LIN {X 0,Y 368.94,Z 360.526,A -85,B 0,C 180,E1 -12835.146,E2 -12835.146} C_VEL
LIN {X 0,Y 368.933,Z 360.527,A -85,B 0,C 180,E1 -12839.046,E2 -12839.046} C_VEL
LIN {X 0,Y 368.972,Z 360.523,A -85,B 0,C 180,E1 -12842.796,E2 -12842.796} C_VEL
LIN {X 0,Y 368.97,Z 360.526,A -85,B 0,C 180,E1 -12846.421,E2 -12846.421} C_VEL
LIN {X 0,Y 368.94,Z 360.529,A -85,B 0,C 180,E1 -12849.946,E2 -12849.946} C_VEL
LIN {X 0,Y 368.979,Z 360.522,A -85,B 0,C 180,E1 -12853.398,E2 -12853.398} C_VEL
LIN {X 0,Y 369.061,Z 360.512,A -85,B 0,C 180,E1 -12856.789,E2 -12856.789} C_VEL
LIN {X 0,Y 369.07,Z 360.514,A -85,B 0,C 180,E1 -12860.131,E2 -12860.131} C_VEL
LIN {X 0,Y 369.201,Z 360.495,A -85,B 0,C 180,E1 -12863.44,E2 -12863.44} C_VEL
LIN {X 0,Y 369.321,Z 360.481,A -85,B 0,C 180,E1 -12867.818,E2 -12867.818} C_VEL
LIN {X 0,Y 369.46,Z 360.465,A -85,B 0,C 180,E1 -12869.999,E2 -12869.999} C_VEL
LIN {X 0,Y 369.32,Z 360.483,A -85,B 0,C 180,E1 -12872.18,E2 -12872.18} C_VEL
LIN {X 0,Y 369.21,Z 360.493,A -85,B 0,C 180,E1 -12876.557,E2 -12876.557} C_VEL
LIN {X 0,Y 369.138,Z 360.501,A -85,B 0,C 180,E1 -12878.76,E2 -12878.76} C_VEL
LIN {X 0,Y 369.006,Z 360.522,A -85,B 0,C 180,E1 -12882.092,E2 -12882.092} C_VEL
LIN {X 0,Y 369,Z 360.52,A -85,B 0,C 180,E1 -12885.463,E2 -12885.463} C_VEL
LIN {X 0,Y 368.981,Z 360.521,A -85,B 0,C 180,E1 -12888.891,E2 -12888.891} C_VEL
LIN {X 0,Y 368.93,Z 360.528,A -85,B 0,C 180,E1 -12892.394,E2 -12892.394} C_VEL
LIN {X 0,Y 368.997,Z 360.524,A -85,B 0,C 180,E1 -12895.979,E2 -12895.979} C_VEL
LIN {X 0,Y 368.964,Z 360.523,A -85,B 0,C 180,E1 -12898.812,E2 -12898.812} C_VEL
LIN {X 0,Y 368.92,Z 360.531,A -85,B 0,C 180,E1 -12899.621,E2 -12899.621} C_VEL
LIN {X 0,Y 368.255,Z 360.62,A -85,B 0,C 180,E1 -12900.532,E2 -12900.532} C_VEL
LIN {X 0,Y 365.401,Z 360.978,A -85,B 0,C 180,E1 -12902.013,E2 -12902.013} C_VEL
LIN {X 0,Y 362.978,Z 361.275,A -85,B 0,C 180,E1 -12903.21,E2 -12903.21} C_VEL
LIN {X 0,Y 361.934,Z 361.401,A -85,B 0,C 180,E1 -12904.137,E2 -12904.137} C_VEL
LIN {X 0,Y 361.846,Z 361.41,A -85,B 0,C 180,E1 -12904.451,E2 -12904.451} C_VEL
LIN {X 0,Y 361.867,Z 361.408,A -85,B 0,C 180,E1 -12907.224,E2 -12907.224} C_VEL
LIN {X 0,Y 361.899,Z 361.402,A -85,B 0,C 180,E1 -12910.767,E2 -12910.767} C_VEL
LIN {X 0,Y 361.927,Z 361.4,A -85,B 0,C 180,E1 -12914.349,E2 -12914.349} C_VEL
LIN {X 0,Y 361.885,Z 361.408,A -85,B 0,C 180,E1 -12917.557,E2 -12917.557} C_VEL
LIN {X 0,Y 361.868,Z 361.407,A -85,B 0,C 180,E1 -12920.971,E2 -12920.971} C_VEL
LIN {X 0,Y 361.867,Z 361.406,A -85,B 0,C 180,E1 -12924.654,E2 -12924.654} C_VEL
LIN {X 0,Y 361.829,Z 361.411,A -85,B 0,C 180,E1 -12928.37,E2 -12928.37} C_VEL
LIN {X 0,Y 361.893,Z 361.403,A -85,B 0,C 180,E1 -12930.955,E2 -12930.955} C_VEL
LIN {X 0,Y 361.946,Z 361.4,A -85,B 0,C 180,E1 -12933.474,E2 -12933.474} C_VEL
LIN {X 0,Y 361.881,Z 361.406,A -85,B 0,C 180,E1 -12937.144,E2 -12937.144} C_VEL
LIN {X 0,Y 361.912,Z 361.4,A -85,B 0,C 180,E1 -12940.724,E2 -12940.724} C_VEL
LIN {X 0,Y 361.939,Z 361.398,A -85,B 0,C 180,E1 -12944.226,E2 -12944.226} C_VEL
LIN {X 0,Y 361.99,Z 361.391,A -85,B 0,C 180,E1 -12946.528,E2 -12946.528} C_VEL
LIN {X 0,Y 362.026,Z 361.389,A -85,B 0,C 180,E1 -12949.938,E2 -12949.938} C_VEL
LIN {X 0,Y 362.141,Z 361.372,A -85,B 0,C 180,E1 -12952.192,E2 -12952.192} C_VEL
LIN {X 0,Y 362.109,Z 361.376,A -85,B 0,C 180,E1 -12954.431,E2 -12954.431} C_VEL
LIN {X 0,Y 362.274,Z 361.359,A -85,B 0,C 180,E1 -12957.777,E2 -12957.777} C_VEL
LIN {X 0,Y 362.42,Z 361.338,A -85,B 0,C 180,E1 -12960,E2 -12960} C_VEL
LIN {X 0,Y 362.274,Z 361.355,A -85,B 0,C 180,E1 -12962.224,E2 -12962.224} C_VEL
LIN {X 0,Y 362.168,Z 361.368,A -85,B 0,C 180,E1 -12966.686,E2 -12966.686} C_VEL
LIN {X 0,Y 362.066,Z 361.382,A -85,B 0,C 180,E1 -12968.934,E2 -12968.934} C_VEL
LIN {X 0,Y 361.958,Z 361.394,A -85,B 0,C 180,E1 -12972.333,E2 -12972.333} C_VEL
LIN {X 0,Y 361.953,Z 361.395,A -85,B 0,C 180,E1 -12974.621,E2 -12974.621} C_VEL
LIN {X 0,Y 361.946,Z 361.397,A -85,B 0,C 180,E1 -12978.1,E2 -12978.1} C_VEL
LIN {X 0,Y 361.884,Z 361.407,A -85,B 0,C 180,E1 -12981.654,E2 -12981.654} C_VEL
LIN {X 0,Y 361.92,Z 361.405,A -85,B 0,C 180,E1 -12985.291,E2 -12985.291} C_VEL
LIN {X 0,Y 361.9,Z 361.404,A -85,B 0,C 180,E1 -12987.78,E2 -12987.78} C_VEL
LIN {X 0,Y 361.83,Z 361.414,A -85,B 0,C 180,E1 -12991.63,E2 -12991.63} C_VEL
LIN {X 0,Y 361.868,Z 361.411,A -85,B 0,C 180,E1 -12995.346,E2 -12995.346} C_VEL
LIN {X 0,Y 361.871,Z 361.409,A -85,B 0,C 180,E1 -12999.029,E2 -12999.029} C_VEL
LIN {X 0,Y 361.881,Z 361.405,A -85,B 0,C 180,E1 -13002.442,E2 -13002.442} C_VEL
LIN {X 0,Y 361.923,Z 361.4,A -85,B 0,C 180,E1 -13005.93,E2 -13005.93} C_VEL
LIN {X 0,Y 361.9,Z 361.407,A -85,B 0,C 180,E1 -13009.233,E2 -13009.233} C_VEL
LIN {X 0,Y 361.866,Z 361.411,A -85,B 0,C 180,E1 -13012.984,E2 -13012.984} C_VEL
LIN {X 0,Y 361.86,Z 361.408,A -85,B 0,C 180,E1 -13016.631,E2 -13016.631} C_VEL
LIN {X 0,Y 361.932,Z 361.44,A -85,B 0,C 180,E1 -13018.647,E2 -13018.647} C_VEL
LIN {X 0,Y 364.497,Z 373.983,A -85,B 0,C 180,E1 -13021.476,E2 -13021.476} C_VEL
LIN {X 0,Y 366.01,Z 381.75,A -85,B 0,C 180,E1 -13023.178,E2 -13023.178} C_VEL
LIN {X 0,Y 364.927,Z 394.849,A -85,B 0,C 180,E1 -13025.844,E2 -13025.844} C_VEL
LIN {X 0,Y 363.607,Z 410.746,A -85,B 0,C 180,E1 -13029.05,E2 -13029.05} C_VEL
LIN {X 0,Y 367.457,Z 446.007,A -85,B 0,C 180,E1 -13030.155,E2 -13030.155} C_VEL
LIN {X 0,Y 365.801,Z 521.346,A -85,B 0,C 180,E1 -13032.135,E2 -13032.135} C_VEL
LIN {X 0,Y 365.107,Z 534.937,A -85,B 0,C 180,E1 -13032.714,E2 -13032.714} C_VEL
LIN {X 0,Y 364.398,Z 547.392,A -85,B 0,C 180,E1 -13033.474,E2 -13033.474} C_VEL
LIN {X 0,Y 363.551,Z 559.509,A -85,B 0,C 180,E1 -13034.443,E2 -13034.443} C_VEL
LIN {X 0,Y 362.806,Z 570.406,A -85,B 0,C 180,E1 -13035.543,E2 -13035.543} C_VEL
LIN {X 0,Y 362.189,Z 580.584,A -85,B 0,C 180,E1 -13036.822,E2 -13036.822} C_VEL
LIN {X 0,Y 361.598,Z 589.732,A -85,B 0,C 180,E1 -13038.226,E2 -13038.226} C_VEL
LIN {X 0,Y 361.106,Z 597.267,A -85,B 0,C 180,E1 -13039.63,E2 -13039.63} C_VEL
LIN {X 0,Y 360.81,Z 604.649,A -85,B 0,C 180,E1 -13041.319,E2 -13041.319} C_VEL
LIN {X 0,Y 360.651,Z 611.306,A -85,B 0,C 180,E1 -13043.287,E2 -13043.287} C_VEL
LIN {X 0,Y 360.631,Z 615.618,A -85,B 0,C 180,E1 -13044.97,E2 -13044.97} C_VEL
LIN {X 0,Y 360.715,Z 618.758,A -85,B 0,C 180,E1 -13046.65,E2 -13046.65} C_VEL
LIN {X 0,Y 360.703,Z 620.246,A -85,B 0,C 180,E1 -13047.768,E2 -13047.768} C_VEL
LIN {X 0,Y 360.8,Z 621.244,A -85,B 0,C 180,E1 -13048.885,E2 -13048.885} C_VEL
LIN {X 0,Y 360.771,Z 621.793,A -85,B 0,C 180,E1 -13050.001,E2 -13050.001} C_VEL
LIN {X 0,Y 360.669,Z 621.901,A -85,B 0,C 180,E1 -13051.118,E2 -13051.118} C_VEL
LIN {X 0,Y 360.653,Z 621.528,A -85,B 0,C 180,E1 -13052.235,E2 -13052.235} C_VEL
LIN {X 0,Y 360.519,Z 620.704,A -85,B 0,C 180,E1 -13053.354,E2 -13053.354} C_VEL
LIN {X 0,Y 360.5,Z 619.46,A -85,B 0,C 180,E1 -13054.474,E2 -13054.474} C_VEL
LIN {X 0,Y 360.521,Z 616.684,A -85,B 0,C 180,E1 -13056.174,E2 -13056.174} C_VEL
LIN {X 0,Y 360.617,Z 612.909,A -85,B 0,C 180,E1 -13057.842,E2 -13057.842} C_VEL
LIN {X 0,Y 360.895,Z 607.954,A -85,B 0,C 180,E1 -13059.529,E2 -13059.529} C_VEL
LIN {X 0,Y 361.418,Z 601.739,A -85,B 0,C 180,E1 -13061.214,E2 -13061.214} C_VEL
LIN {X 0,Y 362.229,Z 594.021,A -85,B 0,C 180,E1 -13062.894,E2 -13062.894} C_VEL
LIN {X 0,Y 363.37,Z 584.53,A -85,B 0,C 180,E1 -13064.564,E2 -13064.564} C_VEL
LIN {X 0,Y 364.563,Z 574.903,A -85,B 0,C 180,E1 -13065.946,E2 -13065.946} C_VEL
LIN {X 0,Y 366.12,Z 563.036,A -85,B 0,C 180,E1 -13067.311,E2 -13067.311} C_VEL
LIN {X 0,Y 367.476,Z 551.355,A -85,B 0,C 180,E1 -13068.396,E2 -13068.396} C_VEL
LIN {X 0,Y 368.985,Z 537.244,A -85,B 0,C 180,E1 -13069.399,E2 -13069.399} C_VEL
LIN {X 0,Y 370.365,Z 524.056,A -85,B 0,C 180,E1 -13070.082,E2 -13070.082} C_VEL
LIN {X 0,Y 371.287,Z 509.676,A -85,B 0,C 180,E1 -13070.608,E2 -13070.608} C_VEL
LIN {X 0,Y 374.2,Z 448.679,A -85,B 0,C 180,E1 -13072.399,E2 -13072.399} C_VEL
LIN {X 0,Y 372.652,Z 431.533,A -85,B 0,C 180,E1 -13073.183,E2 -13073.183} C_VEL
LIN {X 0,Y 370.005,Z 415.628,A -85,B 0,C 180,E1 -13074.086,E2 -13074.086} C_VEL
LIN {X 0,Y 367.095,Z 402.289,A -85,B 0,C 180,E1 -13074.979,E2 -13074.979} C_VEL
LIN {X 0,Y 369.039,Z 390.241,A -85,B 0,C 180,E1 -13077.814,E2 -13077.814} C_VEL
LIN {X 0,Y 367.924,Z 383.506,A -85,B 0,C 180,E1 -13079.78,E2 -13079.78} C_VEL
LIN {X 0,Y 365.968,Z 375.281,A -85,B 0,C 180,E1 -13082.529,E2 -13082.529} C_VEL
LIN {X 0,Y 364.447,Z 369.762,A -85,B 0,C 180,E1 -13084.673,E2 -13084.673} C_VEL
LIN {X 0,Y 363.509,Z 366.42,A -85,B 0,C 180,E1 -13086.135,E2 -13086.135} C_VEL
LIN {X 0,Y 361.879,Z 361.41,A -85,B 0,C 180,E1 -13088.777,E2 -13088.777} C_VEL
LIN {X 0,Y 361.841,Z 361.412,A -85,B 0,C 180,E1 -13092.432,E2 -13092.432} C_VEL
LIN {X 0,Y 361.824,Z 361.415,A -85,B 0,C 180,E1 -13095.947,E2 -13095.947} C_VEL
LIN {X 0,Y 361.841,Z 361.412,A -85,B 0,C 180,E1 -13099.245,E2 -13099.245} C_VEL
LIN {X 0,Y 361.869,Z 361.408,A -85,B 0,C 180,E1 -13102.777,E2 -13102.777} C_VEL
LIN {X 0,Y 361.86,Z 361.409,A -85,B 0,C 180,E1 -13105.72,E2 -13105.72} C_VEL
LIN {X 0,Y 361.88,Z 361.408,A -85,B 0,C 180,E1 -13109.672,E2 -13109.672} C_VEL
LIN {X 0,Y 361.911,Z 361.484,A -85,B 0,C 180,E1 -13110.956,E2 -13110.956} C_VEL
LIN {X 0,Y 363.494,Z 366.94,A -85,B 0,C 180,E1 -13114.213,E2 -13114.213} C_VEL
LIN {X 0,Y 363.789,Z 367.957,A -85,B 0,C 180,E1 -13114.676,E2 -13114.676} C_VEL
LIN {X 0,Y 366.002,Z 371.495,A -85,B 0,C 180,E1 -13115.152,E2 -13115.152} C_VEL
LIN {X 0,Y 372.286,Z 382.279,A -85,B 0,C 180,E1 -13116.436,E2 -13116.436} C_VEL
LIN {X 0,Y 376.514,Z 390.882,A -85,B 0,C 180,E1 -13117.275,E2 -13117.275} C_VEL
LIN {X 0,Y 372.166,Z 469.841,A -85,B 0,C 180,E1 -13119.66,E2 -13119.66} C_VEL
LIN {X 0,Y 371.384,Z 483.921,A -85,B 0,C 180,E1 -13120.301,E2 -13120.301} C_VEL
LIN {X 0,Y 370.566,Z 495.784,A -85,B 0,C 180,E1 -13121.047,E2 -13121.047} C_VEL
LIN {X 0,Y 369.483,Z 507.982,A -85,B 0,C 180,E1 -13122.052,E2 -13122.052} C_VEL
LIN {X 0,Y 368.267,Z 519.085,A -85,B 0,C 180,E1 -13123.2,E2 -13123.2} C_VEL
LIN {X 0,Y 366.989,Z 528.839,A -85,B 0,C 180,E1 -13124.448,E2 -13124.448} C_VEL
LIN {X 0,Y 365.785,Z 537.56,A -85,B 0,C 180,E1 -13125.82,E2 -13125.82} C_VEL
LIN {X 0,Y 364.686,Z 546.093,A -85,B 0,C 180,E1 -13127.479,E2 -13127.479} C_VEL
LIN {X 0,Y 363.741,Z 551.879,A -85,B 0,C 180,E1 -13128.859,E2 -13128.859} C_VEL
LIN {X 0,Y 362.935,Z 557.505,A -85,B 0,C 180,E1 -13130.526,E2 -13130.526} C_VEL
LIN {X 0,Y 362.096,Z 561.9,A -85,B 0,C 180,E1 -13132.191,E2 -13132.191} C_VEL
LIN {X 0,Y 361.868,Z 564.151,A -85,B 0,C 180,E1 -13133.308,E2 -13133.308} C_VEL
LIN {X 0,Y 361.578,Z 565.984,A -85,B 0,C 180,E1 -13134.423,E2 -13134.423} C_VEL
LIN {X 0,Y 361.491,Z 567.341,A -85,B 0,C 180,E1 -13135.54,E2 -13135.54} C_VEL
LIN {X 0,Y 361.247,Z 568.256,A -85,B 0,C 180,E1 -13136.654,E2 -13136.654} C_VEL
LIN {X 0,Y 360.99,Z 568.766,A -85,B 0,C 180,E1 -13137.768,E2 -13137.768} C_VEL
LIN {X 0,Y 360.833,Z 568.854,A -85,B 0,C 180,E1 -13138.884,E2 -13138.884} C_VEL
LIN {X 0,Y 360.723,Z 568.47,A -85,B 0,C 180,E1 -13140,E2 -13140} C_VEL
LIN {X 0,Y 360.696,Z 567.662,A -85,B 0,C 180,E1 -13141.116,E2 -13141.116} C_VEL
LIN {X 0,Y 360.768,Z 566.438,A -85,B 0,C 180,E1 -13142.233,E2 -13142.233} C_VEL
LIN {X 0,Y 360.928,Z 563.739,A -85,B 0,C 180,E1 -13143.908,E2 -13143.908} C_VEL
LIN {X 0,Y 361.008,Z 559.984,A -85,B 0,C 180,E1 -13145.586,E2 -13145.586} C_VEL
LIN {X 0,Y 361.321,Z 554.272,A -85,B 0,C 180,E1 -13147.488,E2 -13147.488} C_VEL
LIN {X 0,Y 361.688,Z 547.573,A -85,B 0,C 180,E1 -13149.225,E2 -13149.225} C_VEL
LIN {X 0,Y 362.225,Z 539.478,A -85,B 0,C 180,E1 -13150.904,E2 -13150.904} C_VEL
LIN {X 0,Y 362.763,Z 531.169,A -85,B 0,C 180,E1 -13152.305,E2 -13152.305} C_VEL
LIN {X 0,Y 363.505,Z 521.067,A -85,B 0,C 180,E1 -13153.7,E2 -13153.7} C_VEL
LIN {X 0,Y 364.212,Z 510.307,A -85,B 0,C 180,E1 -13154.91,E2 -13154.91} C_VEL
LIN {X 0,Y 364.712,Z 498.913,A -85,B 0,C 180,E1 -13155.938,E2 -13155.938} C_VEL
LIN {X 0,Y 365.331,Z 486.039,A -85,B 0,C 180,E1 -13156.844,E2 -13156.844} C_VEL
LIN {X 0,Y 365.926,Z 473.303,A -85,B 0,C 180,E1 -13157.499,E2 -13157.499} C_VEL
LIN {X 0,Y 366.226,Z 460.529,A -85,B 0,C 180,E1 -13157.953,E2 -13157.953} C_VEL
LIN {X 0,Y 368.094,Z 380.127,A -85,B 0,C 180,E1 -13160.016,E2 -13160.016} C_VEL
LIN {X 0,Y 361.937,Z 361.401,A -85,B 0,C 180,E1 -13160.798,E2 -13160.798} C_VEL
LIN {X 0,Y 361.901,Z 361.407,A -85,B 0,C 180,E1 -13164.113,E2 -13164.113} C_VEL
LIN {X 0,Y 361.946,Z 361.4,A -85,B 0,C 180,E1 -13166.721,E2 -13166.721} C_VEL
LIN {X 0,Y 361.88,Z 361.409,A -85,B 0,C 180,E1 -13170.327,E2 -13170.327} C_VEL
LIN {X 0,Y 361.859,Z 361.412,A -85,B 0,C 180,E1 -13174.28,E2 -13174.28} C_VEL
LIN {X 0,Y 361.868,Z 361.407,A -85,B 0,C 180,E1 -13177.222,E2 -13177.222} C_VEL
LIN {X 0,Y 361.84,Z 361.412,A -85,B 0,C 180,E1 -13180.755,E2 -13180.755} C_VEL
LIN {X 0,Y 361.822,Z 361.417,A -85,B 0,C 180,E1 -13184.368,E2 -13184.368} C_VEL
LIN {X 0,Y 361.84,Z 361.411,A -85,B 0,C 180,E1 -13187.567,E2 -13187.567} C_VEL
LIN {X 0,Y 361.874,Z 361.407,A -85,B 0,C 180,E1 -13190.973,E2 -13190.973} C_VEL
LIN {X 0,Y 361.878,Z 361.408,A -85,B 0,C 180,E1 -13194.654,E2 -13194.654} C_VEL
LIN {X 0,Y 361.842,Z 361.415,A -85,B 0,C 180,E1 -13198.37,E2 -13198.37} C_VEL
LIN {X 0,Y 361.916,Z 361.405,A -85,B 0,C 180,E1 -13202.22,E2 -13202.22} C_VEL
LIN {X 0,Y 361.932,Z 361.4,A -85,B 0,C 180,E1 -13204.709,E2 -13204.709} C_VEL
LIN {X 0,Y 361.895,Z 361.407,A -85,B 0,C 180,E1 -13208.346,E2 -13208.346} C_VEL
LIN {X 0,Y 361.971,Z 361.398,A -85,B 0,C 180,E1 -13212.06,E2 -13212.06} C_VEL
LIN {X 0,Y 362.001,Z 361.395,A -85,B 0,C 180,E1 -13216.1,E2 -13216.1} C_VEL
LIN {X 0,Y 362.034,Z 361.39,A -85,B 0,C 180,E1 -13219.937,E2 -13219.937} C_VEL
LIN {X 0,Y 362.163,Z 361.37,A -85,B 0,C 180,E1 -13223.312,E2 -13223.312} C_VEL
LIN {X 0,Y 362.285,Z 361.358,A -85,B 0,C 180,E1 -13227.775,E2 -13227.775} C_VEL
LIN {X 0,Y 362.43,Z 361.341,A -85,B 0,C 180,E1 -13229.999,E2 -13229.999} C_VEL
LIN {X 0,Y 362.284,Z 361.359,A -85,B 0,C 180,E1 -13232.222,E2 -13232.222} C_VEL
LIN {X 0,Y 362.173,Z 361.369,A -85,B 0,C 180,E1 -13236.685,E2 -13236.685} C_VEL
LIN {X 0,Y 362.074,Z 361.381,A -85,B 0,C 180,E1 -13238.932,E2 -13238.932} C_VEL
LIN {X 0,Y 361.96,Z 361.397,A -85,B 0,C 180,E1 -13242.331,E2 -13242.331} C_VEL
LIN {X 0,Y 361.962,Z 361.395,A -85,B 0,C 180,E1 -13244.619,E2 -13244.619} C_VEL
LIN {X 0,Y 361.958,Z 361.4,A -85,B 0,C 180,E1 -13248.098,E2 -13248.098} C_VEL
LIN {X 0,Y 361.889,Z 361.407,A -85,B 0,C 180,E1 -13251.651,E2 -13251.651} C_VEL
LIN {X 0,Y 361.925,Z 361.401,A -85,B 0,C 180,E1 -13255.289,E2 -13255.289} C_VEL
LIN {X 0,Y 361.919,Z 361.404,A -85,B 0,C 180,E1 -13257.776,E2 -13257.776} C_VEL
LIN {X 0,Y 361.855,Z 361.411,A -85,B 0,C 180,E1 -13261.626,E2 -13261.626} C_VEL
LIN {X 0,Y 361.846,Z 361.41,A -85,B 0,C 180,E1 -13264.451,E2 -13264.451} C_VEL
LIN {X 0,Y 361.194,Z 361.493,A -85,B 0,C 180,E1 -13265.38,E2 -13265.38} C_VEL
LIN {X 0,Y 358.419,Z 361.836,A -85,B 0,C 180,E1 -13266.893,E2 -13266.893} C_VEL
LIN {X 0,Y 356.028,Z 362.137,A -85,B 0,C 180,E1 -13268.117,E2 -13268.117} C_VEL
LIN {X 0,Y 354.944,Z 362.27,A -85,B 0,C 180,E1 -13269.062,E2 -13269.062} C_VEL
LIN {X 0,Y 354.824,Z 362.286,A -85,B 0,C 180,E1 -13269.382,E2 -13269.382} C_VEL
LIN {X 0,Y 354.836,Z 362.282,A -85,B 0,C 180,E1 -13272.876,E2 -13272.876} C_VEL
LIN {X 0,Y 354.861,Z 362.282,A -85,B 0,C 180,E1 -13276.118,E2 -13276.118} C_VEL
LIN {X 0,Y 354.85,Z 362.282,A -85,B 0,C 180,E1 -13279.188,E2 -13279.188} C_VEL
LIN {X 0,Y 354.802,Z 362.287,A -85,B 0,C 180,E1 -13282.401,E2 -13282.401} C_VEL
LIN {X 0,Y 354.804,Z 362.286,A -85,B 0,C 180,E1 -13284.94,E2 -13284.94} C_VEL
LIN {X 0,Y 354.785,Z 362.289,A -85,B 0,C 180,E1 -13288.404,E2 -13288.404} C_VEL
LIN {X 0,Y 354.845,Z 362.286,A -85,B 0,C 180,E1 -13291.619,E2 -13291.619} C_VEL
LIN {X 0,Y 354.89,Z 362.277,A -85,B 0,C 180,E1 -13294.172,E2 -13294.172} C_VEL
LIN {X 0,Y 354.826,Z 362.287,A -85,B 0,C 180,E1 -13297.893,E2 -13297.893} C_VEL
LIN {X 0,Y 354.913,Z 362.275,A -85,B 0,C 180,E1 -13301.891,E2 -13301.891} C_VEL
LIN {X 0,Y 354.934,Z 362.272,A -85,B 0,C 180,E1 -13305.98,E2 -13305.98} C_VEL
LIN {X 0,Y 354.973,Z 362.269,A -85,B 0,C 180,E1 -13309.736,E2 -13309.736} C_VEL
LIN {X 0,Y 355.104,Z 362.25,A -85,B 0,C 180,E1 -13312.037,E2 -13312.037} C_VEL
LIN {X 0,Y 355.083,Z 362.251,A -85,B 0,C 180,E1 -13314.321,E2 -13314.321} C_VEL
LIN {X 0,Y 355.237,Z 362.236,A -85,B 0,C 180,E1 -13317.732,E2 -13317.732} C_VEL
LIN {X 0,Y 355.39,Z 362.214,A -85,B 0,C 180,E1 -13320,E2 -13320} C_VEL
LIN {X 0,Y 355.237,Z 362.232,A -85,B 0,C 180,E1 -13322.268,E2 -13322.268} C_VEL
LIN {X 0,Y 355.133,Z 362.245,A -85,B 0,C 180,E1 -13326.819,E2 -13326.819} C_VEL
LIN {X 0,Y 355.007,Z 362.263,A -85,B 0,C 180,E1 -13329.113,E2 -13329.113} C_VEL
LIN {X 0,Y 354.918,Z 362.272,A -85,B 0,C 180,E1 -13332.581,E2 -13332.581} C_VEL
LIN {X 0,Y 354.881,Z 362.277,A -85,B 0,C 180,E1 -13336.097,E2 -13336.097} C_VEL
LIN {X 0,Y 354.892,Z 362.275,A -85,B 0,C 180,E1 -13338.473,E2 -13338.473} C_VEL
LIN {X 0,Y 354.827,Z 362.283,A -85,B 0,C 180,E1 -13342.107,E2 -13342.107} C_VEL
LIN {X 0,Y 354.891,Z 362.277,A -85,B 0,C 180,E1 -13345.828,E2 -13345.828} C_VEL
LIN {X 0,Y 354.809,Z 362.288,A -85,B 0,C 180,E1 -13349.683,E2 -13349.683} C_VEL
LIN {X 0,Y 354.798,Z 362.289,A -85,B 0,C 180,E1 -13353.703,E2 -13353.703} C_VEL
LIN {X 0,Y 354.797,Z 362.287,A -85,B 0,C 180,E1 -13356.46,E2 -13356.46} C_VEL
LIN {X 0,Y 354.819,Z 362.288,A -85,B 0,C 180,E1 -13359.425,E2 -13359.425} C_VEL
LIN {X 0,Y 354.836,Z 362.284,A -85,B 0,C 180,E1 -13362.878,E2 -13362.878} C_VEL
LIN {X 0,Y 354.86,Z 362.279,A -85,B 0,C 180,E1 -13366.12,E2 -13366.12} C_VEL
LIN {X 0,Y 354.851,Z 362.286,A -85,B 0,C 180,E1 -13369.19,E2 -13369.19} C_VEL
LIN {X 0,Y 354.805,Z 362.286,A -85,B 0,C 180,E1 -13372.403,E2 -13372.403} C_VEL
LIN {X 0,Y 354.809,Z 362.289,A -85,B 0,C 180,E1 -13374.942,E2 -13374.942} C_VEL
LIN {X 0,Y 354.914,Z 362.354,A -85,B 0,C 180,E1 -13378.435,E2 -13378.435} C_VEL
LIN {X 0,Y 357.644,Z 375.91,A -85,B 0,C 180,E1 -13381.543,E2 -13381.543} C_VEL
LIN {X 0,Y 359.008,Z 383.544,A -85,B 0,C 180,E1 -13383.242,E2 -13383.242} C_VEL
LIN {X 0,Y 357.542,Z 399.5,A -85,B 0,C 180,E1 -13386.546,E2 -13386.546} C_VEL
LIN {X 0,Y 356.625,Z 410.321,A -85,B 0,C 180,E1 -13388.771,E2 -13388.771} C_VEL
LIN {X 0,Y 359.952,Z 441.619,A -85,B 0,C 180,E1 -13389.773,E2 -13389.773} C_VEL
LIN {X 0,Y 360.614,Z 448.7,A -85,B 0,C 180,E1 -13389.993,E2 -13389.993} C_VEL
LIN {X 0,Y 358.866,Z 520.318,A -85,B 0,C 180,E1 -13391.925,E2 -13391.925} C_VEL
LIN {X 0,Y 358.112,Z 533.958,A -85,B 0,C 180,E1 -13392.513,E2 -13392.513} C_VEL
LIN {X 0,Y 357.371,Z 546.517,A -85,B 0,C 180,E1 -13393.286,E2 -13393.286} C_VEL
LIN {X 0,Y 356.543,Z 558.692,A -85,B 0,C 180,E1 -13394.276,E2 -13394.276} C_VEL
LIN {X 0,Y 355.859,Z 568.814,A -85,B 0,C 180,E1 -13395.306,E2 -13395.306} C_VEL
LIN {X 0,Y 355.296,Z 577.809,A -85,B 0,C 180,E1 -13396.416,E2 -13396.416} C_VEL
LIN {X 0,Y 354.654,Z 586.495,A -85,B 0,C 180,E1 -13397.702,E2 -13397.702} C_VEL
LIN {X 0,Y 354.064,Z 595.898,A -85,B 0,C 180,E1 -13399.421,E2 -13399.421} C_VEL
LIN {X 0,Y 353.764,Z 603.461,A -85,B 0,C 180,E1 -13401.145,E2 -13401.145} C_VEL
LIN {X 0,Y 353.6,Z 608.523,A -85,B 0,C 180,E1 -13402.579,E2 -13402.579} C_VEL
LIN {X 0,Y 353.64,Z 613.396,A -85,B 0,C 180,E1 -13404.299,E2 -13404.299} C_VEL
LIN {X 0,Y 353.537,Z 617.003,A -85,B 0,C 180,E1 -13406.012,E2 -13406.012} C_VEL
LIN {X 0,Y 353.641,Z 619.497,A -85,B 0,C 180,E1 -13407.723,E2 -13407.723} C_VEL
LIN {X 0,Y 353.751,Z 620.563,A -85,B 0,C 180,E1 -13408.863,E2 -13408.863} C_VEL
LIN {X 0,Y 353.723,Z 621.153,A -85,B 0,C 180,E1 -13410.001,E2 -13410.001} C_VEL
LIN {X 0,Y 353.598,Z 621.3,A -85,B 0,C 180,E1 -13411.14,E2 -13411.14} C_VEL
LIN {X 0,Y 353.585,Z 621.009,A -85,B 0,C 180,E1 -13412.28,E2 -13412.28} C_VEL
LIN {X 0,Y 353.427,Z 620.222,A -85,B 0,C 180,E1 -13413.421,E2 -13413.421} C_VEL
LIN {X 0,Y 353.425,Z 619.02,A -85,B 0,C 180,E1 -13414.564,E2 -13414.564} C_VEL
LIN {X 0,Y 353.436,Z 616.599,A -85,B 0,C 180,E1 -13416.151,E2 -13416.151} C_VEL
LIN {X 0,Y 353.541,Z 612.636,A -85,B 0,C 180,E1 -13418,E2 -13418} C_VEL
LIN {X 0,Y 353.877,Z 607.785,A -85,B 0,C 180,E1 -13419.72,E2 -13419.72} C_VEL
LIN {X 0,Y 354.432,Z 601.676,A -85,B 0,C 180,E1 -13421.438,E2 -13421.438} C_VEL
LIN {X 0,Y 355.296,Z 594.149,A -85,B 0,C 180,E1 -13423.15,E2 -13423.15} C_VEL
LIN {X 0,Y 356.494,Z 584.82,A -85,B 0,C 180,E1 -13424.851,E2 -13424.851} C_VEL
LIN {X 0,Y 357.784,Z 575.408,A -85,B 0,C 180,E1 -13426.256,E2 -13426.256} C_VEL
LIN {X 0,Y 359.404,Z 563.899,A -85,B 0,C 180,E1 -13427.645,E2 -13427.645} C_VEL
LIN {X 0,Y 360.824,Z 552.594,A -85,B 0,C 180,E1 -13428.748,E2 -13428.748} C_VEL
LIN {X 0,Y 362.259,Z 540.289,A -85,B 0,C 180,E1 -13429.7,E2 -13429.7} C_VEL
LIN {X 0,Y 363.886,Z 526.38,A -85,B 0,C 180,E1 -13430.492,E2 -13430.492} C_VEL
LIN {X 0,Y 364.98,Z 512.773,A -85,B 0,C 180,E1 -13431.055,E2 -13431.055} C_VEL
LIN {X 0,Y 368.241,Z 449.311,A -85,B 0,C 180,E1 -13432.996,E2 -13432.996} C_VEL
LIN {X 0,Y 366.901,Z 433.584,A -85,B 0,C 180,E1 -13433.746,E2 -13433.746} C_VEL
LIN {X 0,Y 364.548,Z 418.59,A -85,B 0,C 180,E1 -13434.629,E2 -13434.629} C_VEL
LIN {X 0,Y 361.256,Z 403.585,A -85,B 0,C 180,E1 -13435.699,E2 -13435.699} C_VEL
LIN {X 0,Y 360.825,Z 401.292,A -85,B 0,C 180,E1 -13435.869,E2 -13435.869} C_VEL
LIN {X 0,Y 362.405,Z 392.34,A -85,B 0,C 180,E1 -13438.044,E2 -13438.044} C_VEL
LIN {X 0,Y 361.081,Z 384.637,A -85,B 0,C 180,E1 -13440.403,E2 -13440.403} C_VEL
LIN {X 0,Y 359.165,Z 376.733,A -85,B 0,C 180,E1 -13443.224,E2 -13443.224} C_VEL
LIN {X 0,Y 357.721,Z 371.454,A -85,B 0,C 180,E1 -13445.419,E2 -13445.419} C_VEL
LIN {X 0,Y 356.168,Z 366.542,A -85,B 0,C 180,E1 -13447.88,E2 -13447.88} C_VEL
LIN {X 0,Y 354.816,Z 362.288,A -85,B 0,C 180,E1 -13450.631,E2 -13450.631} C_VEL
LIN {X 0,Y 354.772,Z 362.293,A -85,B 0,C 180,E1 -13453.897,E2 -13453.897} C_VEL
LIN {X 0,Y 354.8,Z 362.289,A -85,B 0,C 180,E1 -13457.663,E2 -13457.663} C_VEL
LIN {X 0,Y 354.821,Z 362.287,A -85,B 0,C 180,E1 -13460.666,E2 -13460.666} C_VEL
LIN {X 0,Y 354.827,Z 362.284,A -85,B 0,C 180,E1 -13464.301,E2 -13464.301} C_VEL
LIN {X 0,Y 354.792,Z 362.292,A -85,B 0,C 180,E1 -13467.667,E2 -13467.667} C_VEL
LIN {X 0,Y 354.816,Z 362.348,A -85,B 0,C 180,E1 -13469.168,E2 -13469.168} C_VEL
LIN {X 0,Y 356.308,Z 367.21,A -85,B 0,C 180,E1 -13472.575,E2 -13472.575} C_VEL
LIN {X 0,Y 356.866,Z 369.114,A -85,B 0,C 180,E1 -13473.647,E2 -13473.647} C_VEL
LIN {X 0,Y 359.137,Z 372.643,A -85,B 0,C 180,E1 -13474.184,E2 -13474.184} C_VEL
LIN {X 0,Y 364.34,Z 381.112,A -85,B 0,C 180,E1 -13475.34,E2 -13475.34} C_VEL
LIN {X 0,Y 369.124,Z 390.025,A -85,B 0,C 180,E1 -13476.358,E2 -13476.358} C_VEL
LIN {X 0,Y 370.727,Z 393.298,A -85,B 0,C 180,E1 -13476.688,E2 -13476.688} C_VEL
LIN {X 0,Y 366.08,Z 471.113,A -85,B 0,C 180,E1 -13479.123,E2 -13479.123} C_VEL
LIN {X 0,Y 365.191,Z 485.506,A -85,B 0,C 180,E1 -13479.806,E2 -13479.806} C_VEL
LIN {X 0,Y 364.135,Z 498.829,A -85,B 0,C 180,E1 -13480.699,E2 -13480.699} C_VEL
LIN {X 0,Y 362.888,Z 511.37,A -85,B 0,C 180,E1 -13481.803,E2 -13481.803} C_VEL
LIN {X 0,Y 361.338,Z 523.608,A -85,B 0,C 180,E1 -13483.183,E2 -13483.183} C_VEL
LIN {X 0,Y 360.075,Z 532.53,A -85,B 0,C 180,E1 -13484.432,E2 -13484.432} C_VEL
LIN {X 0,Y 358.662,Z 542.141,A -85,B 0,C 180,E1 -13486.111,E2 -13486.111} C_VEL
LIN {X 0,Y 357.507,Z 549.874,A -85,B 0,C 180,E1 -13487.8,E2 -13487.8} C_VEL
LIN {X 0,Y 356.619,Z 555.103,A -85,B 0,C 180,E1 -13489.209,E2 -13489.209} C_VEL
LIN {X 0,Y 355.574,Z 560.961,A -85,B 0,C 180,E1 -13491.218,E2 -13491.218} C_VEL
LIN {X 0,Y 354.981,Z 564.066,A -85,B 0,C 180,E1 -13492.606,E2 -13492.606} C_VEL
LIN {X 0,Y 354.565,Z 566.852,A -85,B 0,C 180,E1 -13494.312,E2 -13494.312} C_VEL
LIN {X 0,Y 354.469,Z 568.11,A -85,B 0,C 180,E1 -13495.451,E2 -13495.451} C_VEL
LIN {X 0,Y 354.217,Z 568.969,A -85,B 0,C 180,E1 -13496.587,E2 -13496.587} C_VEL
LIN {X 0,Y 353.953,Z 569.426,A -85,B 0,C 180,E1 -13497.724,E2 -13497.724} C_VEL
LIN {X 0,Y 353.758,Z 569.425,A -85,B 0,C 180,E1 -13498.862,E2 -13498.862} C_VEL
LIN {X 0,Y 353.648,Z 568.976,A -85,B 0,C 180,E1 -13500,E2 -13500} C_VEL
LIN {X 0,Y 353.626,Z 568.112,A -85,B 0,C 180,E1 -13501.139,E2 -13501.139} C_VEL
LIN {X 0,Y 353.706,Z 566.814,A -85,B 0,C 180,E1 -13502.277,E2 -13502.277} C_VEL
LIN {X 0,Y 353.839,Z 564.008,A -85,B 0,C 180,E1 -13503.986,E2 -13503.986} C_VEL
LIN {X 0,Y 353.956,Z 560.117,A -85,B 0,C 180,E1 -13505.697,E2 -13505.697} C_VEL
LIN {X 0,Y 354.247,Z 554.491,A -85,B 0,C 180,E1 -13507.567,E2 -13507.567} C_VEL
LIN {X 0,Y 354.657,Z 547.404,A -85,B 0,C 180,E1 -13509.409,E2 -13509.409} C_VEL
LIN {X 0,Y 355.213,Z 539.075,A -85,B 0,C 180,E1 -13511.122,E2 -13511.122} C_VEL
LIN {X 0,Y 355.777,Z 530.576,A -85,B 0,C 180,E1 -13512.55,E2 -13512.55} C_VEL
LIN {X 0,Y 356.57,Z 520.253,A -85,B 0,C 180,E1 -13513.972,E2 -13513.972} C_VEL
LIN {X 0,Y 357.237,Z 509.801,A -85,B 0,C 180,E1 -13515.137,E2 -13515.137} C_VEL
LIN {X 0,Y 357.78,Z 497.318,A -85,B 0,C 180,E1 -13516.255,E2 -13516.255} C_VEL
LIN {X 0,Y 358.435,Z 484.945,A -85,B 0,C 180,E1 -13517.104,E2 -13517.104} C_VEL
LIN {X 0,Y 359.015,Z 470.738,A -85,B 0,C 180,E1 -13517.811,E2 -13517.811} C_VEL
LIN {X 0,Y 359.352,Z 457.7,A -85,B 0,C 180,E1 -13518.235,E2 -13518.235} C_VEL
LIN {X 0,Y 361.131,Z 381.354,A -85,B 0,C 180,E1 -13520.251,E2 -13520.251} C_VEL
LIN {X 0,Y 354.857,Z 362.281,A -85,B 0,C 180,E1 -13521.056,E2 -13521.056} C_VEL
LIN {X 0,Y 354.867,Z 362.283,A -85,B 0,C 180,E1 -13524.576,E2 -13524.576} C_VEL
LIN {X 0,Y 354.888,Z 362.277,A -85,B 0,C 180,E1 -13527.096,E2 -13527.096} C_VEL
LIN {X 0,Y 354.859,Z 362.281,A -85,B 0,C 180,E1 -13529.678,E2 -13529.678} C_VEL
LIN {X 0,Y 354.811,Z 362.287,A -85,B 0,C 180,E1 -13533.701,E2 -13533.701} C_VEL
LIN {X 0,Y 354.803,Z 362.291,A -85,B 0,C 180,E1 -13536.459,E2 -13536.459} C_VEL
LIN {X 0,Y 354.829,Z 362.284,A -85,B 0,C 180,E1 -13539.423,E2 -13539.423} C_VEL
LIN {X 0,Y 354.792,Z 362.289,A -85,B 0,C 180,E1 -13542.866,E2 -13542.866} C_VEL
LIN {X 0,Y 354.772,Z 362.295,A -85,B 0,C 180,E1 -13546.103,E2 -13546.103} C_VEL
LIN {X 0,Y 354.792,Z 362.288,A -85,B 0,C 180,E1 -13549.178,E2 -13549.178} C_VEL
LIN {X 0,Y 354.811,Z 362.29,A -85,B 0,C 180,E1 -13552.402,E2 -13552.402} C_VEL
LIN {X 0,Y 354.816,Z 362.286,A -85,B 0,C 180,E1 -13554.94,E2 -13554.94} C_VEL
LIN {X 0,Y 354.797,Z 362.291,A -85,B 0,C 180,E1 -13558.404,E2 -13558.404} C_VEL
LIN {X 0,Y 354.852,Z 362.282,A -85,B 0,C 180,E1 -13561.618,E2 -13561.618} C_VEL
LIN {X 0,Y 354.903,Z 362.279,A -85,B 0,C 180,E1 -13564.172,E2 -13564.172} C_VEL
LIN {X 0,Y 354.838,Z 362.286,A -85,B 0,C 180,E1 -13567.893,E2 -13567.893} C_VEL
LIN {X 0,Y 354.926,Z 362.275,A -85,B 0,C 180,E1 -13571.89,E2 -13571.89} C_VEL
LIN {X 0,Y 354.946,Z 362.273,A -85,B 0,C 180,E1 -13575.98,E2 -13575.98} C_VEL
LIN {X 0,Y 354.981,Z 362.268,A -85,B 0,C 180,E1 -13579.735,E2 -13579.735} C_VEL
LIN {X 0,Y 355.127,Z 362.246,A -85,B 0,C 180,E1 -13583.179,E2 -13583.179} C_VEL
LIN {X 0,Y 355.248,Z 362.235,A -85,B 0,C 180,E1 -13587.731,E2 -13587.731} C_VEL
LIN {X 0,Y 355.399,Z 362.217,A -85,B 0,C 180,E1 -13589.999,E2 -13589.999} C_VEL
LIN {X 0,Y 355.247,Z 362.235,A -85,B 0,C 180,E1 -13592.266,E2 -13592.266} C_VEL
LIN {X 0,Y 355.139,Z 362.245,A -85,B 0,C 180,E1 -13596.818,E2 -13596.818} C_VEL
LIN {X 0,Y 355.015,Z 362.26,A -85,B 0,C 180,E1 -13599.111,E2 -13599.111} C_VEL
LIN {X 0,Y 354.921,Z 362.273,A -85,B 0,C 180,E1 -13602.579,E2 -13602.579} C_VEL
LIN {X 0,Y 354.891,Z 362.28,A -85,B 0,C 180,E1 -13606.094,E2 -13606.094} C_VEL
LIN {X 0,Y 354.905,Z 362.275,A -85,B 0,C 180,E1 -13608.47,E2 -13608.47} C_VEL
LIN {X 0,Y 354.832,Z 362.287,A -85,B 0,C 180,E1 -13612.105,E2 -13612.105} C_VEL
LIN {X 0,Y 354.896,Z 362.28,A -85,B 0,C 180,E1 -13615.826,E2 -13615.826} C_VEL
LIN {X 0,Y 354.85,Z 362.284,A -85,B 0,C 180,E1 -13619.677,E2 -13619.677} C_VEL
LIN {X 0,Y 354.826,Z 362.288,A -85,B 0,C 180,E1 -13623.681,E2 -13623.681} C_VEL
LIN {X 0,Y 354.797,Z 362.288,A -85,B 0,C 180,E1 -13626.458,E2 -13626.458} C_VEL
LIN {X 0,Y 354.824,Z 362.286,A -85,B 0,C 180,E1 -13629.382,E2 -13629.382} C_VEL
LIN {X 0,Y 354.073,Z 362.384,A -85,B 0,C 180,E1 -13630.328,E2 -13630.328} C_VEL
LIN {X 0,Y 351.206,Z 362.74,A -85,B 0,C 180,E1 -13631.868,E2 -13631.868} C_VEL
LIN {X 0,Y 348.846,Z 363.029,A -85,B 0,C 180,E1 -13633.114,E2 -13633.114} C_VEL
LIN {X 0,Y 347.859,Z 363.154,A -85,B 0,C 180,E1 -13634.077,E2 -13634.077} C_VEL
LIN {X 0,Y 347.789,Z 363.157,A -85,B 0,C 180,E1 -13634.403,E2 -13634.403} C_VEL
LIN {X 0,Y 347.811,Z 363.157,A -85,B 0,C 180,E1 -13636.669,E2 -13636.669} C_VEL
LIN {X 0,Y 347.778,Z 363.163,A -85,B 0,C 180,E1 -13640.164,E2 -13640.164} C_VEL
LIN {X 0,Y 347.781,Z 363.163,A -85,B 0,C 180,E1 -13644.124,E2 -13644.124} C_VEL
LIN {X 0,Y 347.731,Z 363.169,A -85,B 0,C 180,E1 -13648.085,E2 -13648.085} C_VEL
LIN {X 0,Y 347.797,Z 363.159,A -85,B 0,C 180,E1 -13650.989,E2 -13650.989} C_VEL
LIN {X 0,Y 347.823,Z 363.161,A -85,B 0,C 180,E1 -13653.607,E2 -13653.607} C_VEL
LIN {X 0,Y 347.779,Z 363.162,A -85,B 0,C 180,E1 -13656.161,E2 -13656.161} C_VEL
LIN {X 0,Y 347.809,Z 363.16,A -85,B 0,C 180,E1 -13659.909,E2 -13659.909} C_VEL
LIN {X 0,Y 347.858,Z 363.151,A -85,B 0,C 180,E1 -13662.359,E2 -13662.359} C_VEL
LIN {X 0,Y 347.888,Z 363.15,A -85,B 0,C 180,E1 -13665.971,E2 -13665.971} C_VEL
LIN {X 0,Y 347.923,Z 363.149,A -85,B 0,C 180,E1 -13669.526,E2 -13669.526} C_VEL
LIN {X 0,Y 348.064,Z 363.128,A -85,B 0,C 180,E1 -13671.875,E2 -13671.875} C_VEL
LIN {X 0,Y 348.058,Z 363.127,A -85,B 0,C 180,E1 -13674.206,E2 -13674.206} C_VEL
LIN {X 0,Y 348.199,Z 363.113,A -85,B 0,C 180,E1 -13677.687,E2 -13677.687} C_VEL
LIN {X 0,Y 348.359,Z 363.09,A -85,B 0,C 180,E1 -13680,E2 -13680} C_VEL
LIN {X 0,Y 348.2,Z 363.108,A -85,B 0,C 180,E1 -13682.314,E2 -13682.314} C_VEL
LIN {X 0,Y 348.1,Z 363.122,A -85,B 0,C 180,E1 -13686.958,E2 -13686.958} C_VEL
LIN {X 0,Y 347.96,Z 363.143,A -85,B 0,C 180,E1 -13689.299,E2 -13689.299} C_VEL
LIN {X 0,Y 347.885,Z 363.149,A -85,B 0,C 180,E1 -13692.84,E2 -13692.84} C_VEL
LIN {X 0,Y 347.83,Z 363.154,A -85,B 0,C 180,E1 -13696.432,E2 -13696.432} C_VEL
LIN {X 0,Y 347.842,Z 363.154,A -85,B 0,C 180,E1 -13698.861,E2 -13698.861} C_VEL
LIN {X 0,Y 347.767,Z 363.163,A -85,B 0,C 180,E1 -13702.58,E2 -13702.58} C_VEL
LIN {X 0,Y 347.804,Z 363.161,A -85,B 0,C 180,E1 -13705.109,E2 -13705.109} C_VEL
LIN {X 0,Y 347.8,Z 363.161,A -85,B 0,C 180,E1 -13707.695,E2 -13707.695} C_VEL
LIN {X 0,Y 347.741,Z 363.166,A -85,B 0,C 180,E1 -13710.349,E2 -13710.349} C_VEL
LIN {X 0,Y 347.741,Z 363.166,A -85,B 0,C 180,E1 -13714.045,E2 -13714.045} C_VEL
LIN {X 0,Y 347.762,Z 363.169,A -85,B 0,C 180,E1 -13717.321,E2 -13717.321} C_VEL
LIN {X 0,Y 347.787,Z 363.16,A -85,B 0,C 180,E1 -13720.29,E2 -13720.29} C_VEL
LIN {X 0,Y 347.813,Z 363.161,A -85,B 0,C 180,E1 -13723.394,E2 -13723.394} C_VEL
LIN {X 0,Y 347.812,Z 363.158,A -85,B 0,C 180,E1 -13726.672,E2 -13726.672} C_VEL
LIN {X 0,Y 347.781,Z 363.161,A -85,B 0,C 180,E1 -13730.167,E2 -13730.167} C_VEL
LIN {X 0,Y 347.786,Z 363.16,A -85,B 0,C 180,E1 -13734.126,E2 -13734.126} C_VEL
LIN {X 0,Y 347.856,Z 363.206,A -85,B 0,C 180,E1 -13738.208,E2 -13738.208} C_VEL
LIN {X 0,Y 350.782,Z 377.668,A -85,B 0,C 180,E1 -13741.588,E2 -13741.588} C_VEL
LIN {X 0,Y 351.959,Z 383.81,A -85,B 0,C 180,E1 -13742.983,E2 -13742.983} C_VEL
LIN {X 0,Y 350.963,Z 395.447,A -85,B 0,C 180,E1 -13745.45,E2 -13745.45} C_VEL
LIN {X 0,Y 349.621,Z 409.861,A -85,B 0,C 180,E1 -13748.48,E2 -13748.48} C_VEL
LIN {X 0,Y 352.958,Z 441.979,A -85,B 0,C 180,E1 -13749.536,E2 -13749.536} C_VEL
LIN {X 0,Y 353.639,Z 449.699,A -85,B 0,C 180,E1 -13749.783,E2 -13749.783} C_VEL
LIN {X 0,Y 351.862,Z 520.021,A -85,B 0,C 180,E1 -13751.741,E2 -13751.741} C_VEL
LIN {X 0,Y 351.136,Z 532.858,A -85,B 0,C 180,E1 -13752.305,E2 -13752.305} C_VEL
LIN {X 0,Y 350.321,Z 545.54,A -85,B 0,C 180,E1 -13753.09,E2 -13753.09} C_VEL
LIN {X 0,Y 349.54,Z 557.798,A -85,B 0,C 180,E1 -13754.102,E2 -13754.102} C_VEL
LIN {X 0,Y 348.726,Z 569.459,A -85,B 0,C 180,E1 -13755.322,E2 -13755.322} C_VEL
LIN {X 0,Y 348.113,Z 579.093,A -85,B 0,C 180,E1 -13756.577,E2 -13756.577} C_VEL
LIN {X 0,Y 347.486,Z 588.304,A -85,B 0,C 180,E1 -13758.037,E2 -13758.037} C_VEL
LIN {X 0,Y 346.901,Z 597.276,A -85,B 0,C 180,E1 -13759.791,E2 -13759.791} C_VEL
LIN {X 0,Y 346.654,Z 604.407,A -85,B 0,C 180,E1 -13761.549,E2 -13761.549} C_VEL
LIN {X 0,Y 346.54,Z 610.873,A -85,B 0,C 180,E1 -13763.59,E2 -13763.59} C_VEL
LIN {X 0,Y 346.452,Z 615.016,A -85,B 0,C 180,E1 -13765.347,E2 -13765.347} C_VEL
LIN {X 0,Y 346.559,Z 617.101,A -85,B 0,C 180,E1 -13766.513,E2 -13766.513} C_VEL
LIN {X 0,Y 346.58,Z 618.709,A -85,B 0,C 180,E1 -13767.677,E2 -13767.677} C_VEL
LIN {X 0,Y 346.703,Z 619.868,A -85,B 0,C 180,E1 -13768.84,E2 -13768.84} C_VEL
LIN {X 0,Y 346.676,Z 620.506,A -85,B 0,C 180,E1 -13770.001,E2 -13770.001} C_VEL
LIN {X 0,Y 346.53,Z 620.696,A -85,B 0,C 180,E1 -13771.163,E2 -13771.163} C_VEL
LIN {X 0,Y 346.517,Z 620.462,A -85,B 0,C 180,E1 -13772.326,E2 -13772.326} C_VEL
LIN {X 0,Y 346.338,Z 619.75,A -85,B 0,C 180,E1 -13773.491,E2 -13773.491} C_VEL
LIN {X 0,Y 346.33,Z 618.587,A -85,B 0,C 180,E1 -13774.657,E2 -13774.657} C_VEL
LIN {X 0,Y 346.331,Z 616.58,A -85,B 0,C 180,E1 -13776.095,E2 -13776.095} C_VEL
LIN {X 0,Y 346.487,Z 612.394,A -85,B 0,C 180,E1 -13778.164,E2 -13778.164} C_VEL
LIN {X 0,Y 346.844,Z 607.651,A -85,B 0,C 180,E1 -13779.919,E2 -13779.919} C_VEL
LIN {X 0,Y 347.458,Z 601.662,A -85,B 0,C 180,E1 -13781.671,E2 -13781.671} C_VEL
LIN {X 0,Y 348.377,Z 594.288,A -85,B 0,C 180,E1 -13783.416,E2 -13783.416} C_VEL
LIN {X 0,Y 349.653,Z 585.194,A -85,B 0,C 180,E1 -13785.148,E2 -13785.148} C_VEL
LIN {X 0,Y 351.021,Z 576.003,A -85,B 0,C 180,E1 -13786.578,E2 -13786.578} C_VEL
LIN {X 0,Y 352.703,Z 564.861,A -85,B 0,C 180,E1 -13787.991,E2 -13787.991} C_VEL
LIN {X 0,Y 354.198,Z 553.981,A -85,B 0,C 180,E1 -13789.112,E2 -13789.112} C_VEL
LIN {X 0,Y 355.936,Z 540.336,A -85,B 0,C 180,E1 -13790.216,E2 -13790.216} C_VEL
LIN {X 0,Y 357.633,Z 526.857,A -85,B 0,C 180,E1 -13791.018,E2 -13791.018} C_VEL
LIN {X 0,Y 358.893,Z 512.151,A -85,B 0,C 180,E1 -13791.656,E2 -13791.656} C_VEL
LIN {X 0,Y 362.418,Z 450.492,A -85,B 0,C 180,E1 -13793.601,E2 -13793.601} C_VEL
LIN {X 0,Y 361.162,Z 434.701,A -85,B 0,C 180,E1 -13794.389,E2 -13794.389} C_VEL
LIN {X 0,Y 358.887,Z 419.888,A -85,B 0,C 180,E1 -13795.311,E2 -13795.311} C_VEL
LIN {X 0,Y 355.464,Z 403.973,A -85,B 0,C 180,E1 -13796.516,E2 -13796.516} C_VEL
LIN {X 0,Y 354.647,Z 400.208,A -85,B 0,C 180,E1 -13796.851,E2 -13796.851} C_VEL
LIN {X 0,Y 355.789,Z 394.42,A -85,B 0,C 180,E1 -13798.301,E2 -13798.301} C_VEL
LIN {X 0,Y 354.493,Z 386.905,A -85,B 0,C 180,E1 -13800.699,E2 -13800.699} C_VEL
LIN {X 0,Y 352.874,Z 380.034,A -85,B 0,C 180,E1 -13803.228,E2 -13803.228} C_VEL
LIN {X 0,Y 351.487,Z 374.848,A -85,B 0,C 180,E1 -13805.442,E2 -13805.442} C_VEL
LIN {X 0,Y 349.717,Z 369.221,A -85,B 0,C 180,E1 -13808.394,E2 -13808.394} C_VEL
LIN {X 0,Y 348.813,Z 366.541,A -85,B 0,C 180,E1 -13810.148,E2 -13810.148} C_VEL
LIN {X 0,Y 347.746,Z 363.168,A -85,B 0,C 180,E1 -13813.09,E2 -13813.09} C_VEL
LIN {X 0,Y 347.731,Z 363.169,A -85,B 0,C 180,E1 -13816.687,E2 -13816.687} C_VEL
LIN {X 0,Y 347.753,Z 363.169,A -85,B 0,C 180,E1 -13820.173,E2 -13820.173} C_VEL
LIN {X 0,Y 347.767,Z 363.164,A -85,B 0,C 180,E1 -13822.68,E2 -13822.68} C_VEL
LIN {X 0,Y 347.781,Z 363.164,A -85,B 0,C 180,E1 -13826.448,E2 -13826.448} C_VEL
LIN {X 0,Y 347.792,Z 363.374,A -85,B 0,C 180,E1 -13826.934,E2 -13826.934} C_VEL
LIN {X 0,Y 348.846,Z 366.823,A -85,B 0,C 180,E1 -13830.033,E2 -13830.033} C_VEL
LIN {X 0,Y 350.01,Z 370.438,A -85,B 0,C 180,E1 -13832.508,E2 -13832.508} C_VEL
LIN {X 0,Y 352.512,Z 374.147,A -85,B 0,C 180,E1 -13833.156,E2 -13833.156} C_VEL
LIN {X 0,Y 357.704,Z 382.164,A -85,B 0,C 180,E1 -13834.414,E2 -13834.414} C_VEL
LIN {X 0,Y 363.071,Z 391.88,A -85,B 0,C 180,E1 -13835.638,E2 -13835.638} C_VEL
LIN {X 0,Y 364.992,Z 396.025,A -85,B 0,C 180,E1 -13836.074,E2 -13836.074} C_VEL
LIN {X 0,Y 360.103,Z 471.941,A -85,B 0,C 180,E1 -13838.535,E2 -13838.535} C_VEL
LIN {X 0,Y 359.146,Z 486.146,A -85,B 0,C 180,E1 -13839.226,E2 -13839.226} C_VEL
LIN {X 0,Y 358.11,Z 498.5,A -85,B 0,C 180,E1 -13840.063,E2 -13840.063} C_VEL
LIN {X 0,Y 356.928,Z 509.745,A -85,B 0,C 180,E1 -13841.042,E2 -13841.042} C_VEL
LIN {X 0,Y 355.56,Z 520.513,A -85,B 0,C 180,E1 -13842.204,E2 -13842.204} C_VEL
LIN {X 0,Y 354.006,Z 530.705,A -85,B 0,C 180,E1 -13843.566,E2 -13843.566} C_VEL
LIN {X 0,Y 352.634,Z 539.302,A -85,B 0,C 180,E1 -13844.984,E2 -13844.984} C_VEL
LIN {X 0,Y 351.326,Z 547.71,A -85,B 0,C 180,E1 -13846.7,E2 -13846.7} C_VEL
LIN {X 0,Y 350.089,Z 554.421,A -85,B 0,C 180,E1 -13848.419,E2 -13848.419} C_VEL
LIN {X 0,Y 349.15,Z 559.752,A -85,B 0,C 180,E1 -13850.148,E2 -13850.148} C_VEL
LIN {X 0,Y 348.196,Z 563.901,A -85,B 0,C 180,E1 -13851.877,E2 -13851.877} C_VEL
LIN {X 0,Y 347.887,Z 566.042,A -85,B 0,C 180,E1 -13853.038,E2 -13853.038} C_VEL
LIN {X 0,Y 347.555,Z 567.704,A -85,B 0,C 180,E1 -13854.197,E2 -13854.197} C_VEL
LIN {X 0,Y 347.448,Z 568.892,A -85,B 0,C 180,E1 -13855.359,E2 -13855.359} C_VEL
LIN {X 0,Y 347.189,Z 569.694,A -85,B 0,C 180,E1 -13856.518,E2 -13856.518} C_VEL
LIN {X 0,Y 346.917,Z 570.075,A -85,B 0,C 180,E1 -13857.678,E2 -13857.678} C_VEL
LIN {X 0,Y 346.685,Z 569.987,A -85,B 0,C 180,E1 -13858.838,E2 -13858.838} C_VEL
LIN {X 0,Y 346.575,Z 569.479,A -85,B 0,C 180,E1 -13860,E2 -13860} C_VEL
LIN {X 0,Y 346.559,Z 568.553,A -85,B 0,C 180,E1 -13861.162,E2 -13861.162} C_VEL
LIN {X 0,Y 346.646,Z 567.149,A -85,B 0,C 180,E1 -13862.324,E2 -13862.324} C_VEL
LIN {X 0,Y 346.748,Z 564.222,A -85,B 0,C 180,E1 -13864.068,E2 -13864.068} C_VEL
LIN {X 0,Y 346.882,Z 560.202,A -85,B 0,C 180,E1 -13865.814,E2 -13865.814} C_VEL
LIN {X 0,Y 347.208,Z 553.996,A -85,B 0,C 180,E1 -13867.852,E2 -13867.852} C_VEL
LIN {X 0,Y 347.614,Z 547.161,A -85,B 0,C 180,E1 -13869.602,E2 -13869.602} C_VEL
LIN {X 0,Y 348.218,Z 538.627,A -85,B 0,C 180,E1 -13871.349,E2 -13871.349} C_VEL
LIN {X 0,Y 348.812,Z 529.929,A -85,B 0,C 180,E1 -13872.805,E2 -13872.805} C_VEL
LIN {X 0,Y 349.555,Z 519.245,A -85,B 0,C 180,E1 -13874.258,E2 -13874.258} C_VEL
LIN {X 0,Y 350.35,Z 507.206,A -85,B 0,C 180,E1 -13875.571,E2 -13875.571} C_VEL
LIN {X 0,Y 350.902,Z 495.446,A -85,B 0,C 180,E1 -13876.583,E2 -13876.583} C_VEL
LIN {X 0,Y 351.563,Z 482.306,A -85,B 0,C 180,E1 -13877.449,E2 -13877.449} C_VEL
LIN {X 0,Y 352.033,Z 469.433,A -85,B 0,C 180,E1 -13878.063,E2 -13878.063} C_VEL
LIN {X 0,Y 352.49,Z 448.912,A -85,B 0,C 180,E1 -13878.678,E2 -13878.678} C_VEL
LIN {X 0,Y 354.211,Z 382.777,A -85,B 0,C 180,E1 -13880.485,E2 -13880.485} C_VEL
LIN {X 0,Y 347.83,Z 363.155,A -85,B 0,C 180,E1 -13881.327,E2 -13881.327} C_VEL
LIN {X 0,Y 347.817,Z 363.157,A -85,B 0,C 180,E1 -13885.108,E2 -13885.108} C_VEL
LIN {X 0,Y 347.815,Z 363.158,A -85,B 0,C 180,E1 -13887.693,E2 -13887.693} C_VEL
LIN {X 0,Y 347.769,Z 363.167,A -85,B 0,C 180,E1 -13890.346,E2 -13890.346} C_VEL
LIN {X 0,Y 347.749,Z 363.17,A -85,B 0,C 180,E1 -13894.463,E2 -13894.463} C_VEL
LIN {X 0,Y 347.778,Z 363.165,A -85,B 0,C 180,E1 -13897.988,E2 -13897.988} C_VEL
LIN {X 0,Y 347.755,Z 363.167,A -85,B 0,C 180,E1 -13901.83,E2 -13901.83} C_VEL
LIN {X 0,Y 347.71,Z 363.17,A -85,B 0,C 180,E1 -13905.026,E2 -13905.026} C_VEL
LIN {X 0,Y 347.755,Z 363.169,A -85,B 0,C 180,E1 -13908.396,E2 -13908.396} C_VEL
LIN {X 0,Y 347.778,Z 363.166,A -85,B 0,C 180,E1 -13912.01,E2 -13912.01} C_VEL
LIN {X 0,Y 347.748,Z 363.166,A -85,B 0,C 180,E1 -13915.535,E2 -13915.535} C_VEL
LIN {X 0,Y 347.749,Z 363.17,A -85,B 0,C 180,E1 -13918.3,E2 -13918.3} C_VEL
LIN {X 0,Y 347.783,Z 363.161,A -85,B 0,C 180,E1 -13920.987,E2 -13920.987} C_VEL
LIN {X 0,Y 347.835,Z 363.156,A -85,B 0,C 180,E1 -13923.607,E2 -13923.607} C_VEL
LIN {X 0,Y 347.792,Z 363.165,A -85,B 0,C 180,E1 -13926.161,E2 -13926.161} C_VEL
LIN {X 0,Y 347.821,Z 363.16,A -85,B 0,C 180,E1 -13929.909,E2 -13929.909} C_VEL
LIN {X 0,Y 347.87,Z 363.154,A -85,B 0,C 180,E1 -13932.358,E2 -13932.358} C_VEL
LIN {X 0,Y 347.9,Z 363.151,A -85,B 0,C 180,E1 -13935.97,E2 -13935.97} C_VEL
LIN {X 0,Y 347.931,Z 363.144,A -85,B 0,C 180,E1 -13939.524,E2 -13939.524} C_VEL
LIN {X 0,Y 348.093,Z 363.122,A -85,B 0,C 180,E1 -13943.041,E2 -13943.041} C_VEL
LIN {X 0,Y 348.21,Z 363.111,A -85,B 0,C 180,E1 -13947.685,E2 -13947.685} C_VEL
LIN {X 0,Y 348.369,Z 363.093,A -85,B 0,C 180,E1 -13949.999,E2 -13949.999} C_VEL
LIN {X 0,Y 348.21,Z 363.111,A -85,B 0,C 180,E1 -13952.312,E2 -13952.312} C_VEL
LIN {X 0,Y 348.107,Z 363.12,A -85,B 0,C 180,E1 -13956.956,E2 -13956.956} C_VEL
LIN {X 0,Y 347.967,Z 363.139,A -85,B 0,C 180,E1 -13959.297,E2 -13959.297} C_VEL
LIN {X 0,Y 347.89,Z 363.148,A -85,B 0,C 180,E1 -13962.838,E2 -13962.838} C_VEL
LIN {X 0,Y 347.84,Z 363.155,A -85,B 0,C 180,E1 -13966.43,E2 -13966.43} C_VEL
LIN {X 0,Y 347.854,Z 363.152,A -85,B 0,C 180,E1 -13968.859,E2 -13968.859} C_VEL
LIN {X 0,Y 347.772,Z 363.163,A -85,B 0,C 180,E1 -13972.578,E2 -13972.578} C_VEL
LIN {X 0,Y 347.809,Z 363.158,A -85,B 0,C 180,E1 -13975.107,E2 -13975.107} C_VEL
LIN {X 0,Y 347.809,Z 363.162,A -85,B 0,C 180,E1 -13977.692,E2 -13977.692} C_VEL
LIN {X 0,Y 347.766,Z 363.164,A -85,B 0,C 180,E1 -13980.344,E2 -13980.344} C_VEL
LIN {X 0,Y 347.743,Z 363.169,A -85,B 0,C 180,E1 -13984.043,E2 -13984.043} C_VEL
LIN {X 0,Y 347.762,Z 363.165,A -85,B 0,C 180,E1 -13987.319,E2 -13987.319} C_VEL
LIN {X 0,Y 347.787,Z 363.162,A -85,B 0,C 180,E1 -13990.287,E2 -13990.287} C_VEL
LIN {X 0,Y 347.813,Z 363.159,A -85,B 0,C 180,E1 -13993.392,E2 -13993.392} C_VEL
LIN {X 0,Y 347.789,Z 363.157,A -85,B 0,C 180,E1 -13994.403,E2 -13994.403} C_VEL
LIN {X 0,Y 347.135,Z 363.245,A -85,B 0,C 180,E1 -13995.37,E2 -13995.37} C_VEL
LIN {X 0,Y 344.247,Z 363.601,A -85,B 0,C 180,E1 -13996.942,E2 -13996.942} C_VEL
LIN {X 0,Y 341.812,Z 363.906,A -85,B 0,C 180,E1 -13998.215,E2 -13998.215} C_VEL
LIN {X 0,Y 340.803,Z 364.031,A -85,B 0,C 180,E1 -13999.201,E2 -13999.201} C_VEL
LIN {X 0,Y 340.741,Z 364.041,A -85,B 0,C 180,E1 -13999.535,E2 -13999.535} C_VEL
LIN {X 0,Y 340.698,Z 364.045,A -85,B 0,C 180,E1 -14003.258,E2 -14003.258} C_VEL
LIN {X 0,Y 340.686,Z 364.046,A -85,B 0,C 180,E1 -14006.153,E2 -14006.153} C_VEL
LIN {X 0,Y 340.766,Z 364.035,A -85,B 0,C 180,E1 -14010.332,E2 -14010.332} C_VEL
LIN {X 0,Y 340.796,Z 364.032,A -85,B 0,C 180,E1 -14013.019,E2 -14013.019} C_VEL
LIN {X 0,Y 340.719,Z 364.041,A -85,B 0,C 180,E1 -14016.927,E2 -14016.927} C_VEL
LIN {X 0,Y 340.786,Z 364.032,A -85,B 0,C 180,E1 -14020.733,E2 -14020.733} C_VEL
LIN {X 0,Y 340.779,Z 364.035,A -85,B 0,C 180,E1 -14023.218,E2 -14023.218} C_VEL
LIN {X 0,Y 340.837,Z 364.026,A -85,B 0,C 180,E1 -14026.89,E2 -14026.89} C_VEL
LIN {X 0,Y 340.92,Z 364.015,A -85,B 0,C 180,E1 -14030.508,E2 -14030.508} C_VEL
LIN {X 0,Y 341.066,Z 363.998,A -85,B 0,C 180,E1 -14032.898,E2 -14032.898} C_VEL
LIN {X 0,Y 341.161,Z 363.99,A -85,B 0,C 180,E1 -14037.639,E2 -14037.639} C_VEL
LIN {X 0,Y 341.308,Z 363.968,A -85,B 0,C 180,E1 -14040,E2 -14040} C_VEL
LIN {X 0,Y 341.162,Z 363.985,A -85,B 0,C 180,E1 -14042.361,E2 -14042.361} C_VEL
LIN {X 0,Y 341.069,Z 363.999,A -85,B 0,C 180,E1 -14047.102,E2 -14047.102} C_VEL
LIN {X 0,Y 340.866,Z 364.022,A -85,B 0,C 180,E1 -14050.694,E2 -14050.694} C_VEL
LIN {X 0,Y 340.854,Z 364.023,A -85,B 0,C 180,E1 -14054.325,E2 -14054.325} C_VEL
LIN {X 0,Y 340.828,Z 364.027,A -85,B 0,C 180,E1 -14058.467,E2 -14058.467} C_VEL
LIN {X 0,Y 340.745,Z 364.039,A -85,B 0,C 180,E1 -14061.858,E2 -14061.858} C_VEL
LIN {X 0,Y 340.764,Z 364.038,A -85,B 0,C 180,E1 -14065.665,E2 -14065.665} C_VEL
LIN {X 0,Y 340.72,Z 364.04,A -85,B 0,C 180,E1 -14068.322,E2 -14068.322} C_VEL
LIN {X 0,Y 340.69,Z 364.047,A -85,B 0,C 180,E1 -14071.046,E2 -14071.046} C_VEL
LIN {X 0,Y 340.712,Z 364.047,A -85,B 0,C 180,E1 -14075.28,E2 -14075.28} C_VEL
LIN {X 0,Y 340.719,Z 364.04,A -85,B 0,C 180,E1 -14078.391,E2 -14078.391} C_VEL
LIN {X 0,Y 340.746,Z 364.037,A -85,B 0,C 180,E1 -14082.057,E2 -14082.057} C_VEL
LIN {X 0,Y 340.776,Z 364.037,A -85,B 0,C 180,E1 -14085.479,E2 -14085.479} C_VEL
LIN {X 0,Y 340.721,Z 364.042,A -85,B 0,C 180,E1 -14088.698,E2 -14088.698} C_VEL
LIN {X 0,Y 340.735,Z 364.04,A -85,B 0,C 180,E1 -14091.775,E2 -14091.775} C_VEL
LIN {X 0,Y 340.719,Z 364.043,A -85,B 0,C 180,E1 -14095.597,E2 -14095.597} C_VEL
LIN {X 0,Y 340.779,Z 364.197,A -85,B 0,C 180,E1 -14098.011,E2 -14098.011} C_VEL
LIN {X 0,Y 343.44,Z 377.181,A -85,B 0,C 180,E1 -14101.117,E2 -14101.117} C_VEL
LIN {X 0,Y 344.967,Z 385.511,A -85,B 0,C 180,E1 -14103.046,E2 -14103.046} C_VEL
LIN {X 0,Y 343.368,Z 401.419,A -85,B 0,C 180,E1 -14106.478,E2 -14106.478} C_VEL
LIN {X 0,Y 342.65,Z 409.345,A -85,B 0,C 180,E1 -14108.178,E2 -14108.178} C_VEL
LIN {X 0,Y 345.751,Z 440.326,A -85,B 0,C 180,E1 -14109.234,E2 -14109.234} C_VEL
LIN {X 0,Y 346.738,Z 449.104,A -85,B 0,C 180,E1 -14109.527,E2 -14109.527} C_VEL
LIN {X 0,Y 344.869,Z 519.392,A -85,B 0,C 180,E1 -14111.55,E2 -14111.55} C_VEL
LIN {X 0,Y 344.104,Z 532.875,A -85,B 0,C 180,E1 -14112.162,E2 -14112.162} C_VEL
LIN {X 0,Y 343.324,Z 544.387,A -85,B 0,C 180,E1 -14112.888,E2 -14112.888} C_VEL
LIN {X 0,Y 342.56,Z 556.781,A -85,B 0,C 180,E1 -14113.922,E2 -14113.922} C_VEL
LIN {X 0,Y 341.693,Z 568.607,A -85,B 0,C 180,E1 -14115.174,E2 -14115.174} C_VEL
LIN {X 0,Y 341.075,Z 578.249,A -85,B 0,C 180,E1 -14116.446,E2 -14116.446} C_VEL
LIN {X 0,Y 340.371,Z 588.354,A -85,B 0,C 180,E1 -14118.085,E2 -14118.085} C_VEL
LIN {X 0,Y 339.875,Z 595.852,A -85,B 0,C 180,E1 -14119.577,E2 -14119.577} C_VEL
LIN {X 0,Y 339.592,Z 603.182,A -85,B 0,C 180,E1 -14121.372,E2 -14121.372} C_VEL
LIN {X 0,Y 339.453,Z 609.141,A -85,B 0,C 180,E1 -14123.228,E2 -14123.228} C_VEL
LIN {X 0,Y 339.478,Z 612.792,A -85,B 0,C 180,E1 -14124.656,E2 -14124.656} C_VEL
LIN {X 0,Y 339.487,Z 616.24,A -85,B 0,C 180,E1 -14126.441,E2 -14126.441} C_VEL
LIN {X 0,Y 339.52,Z 617.901,A -85,B 0,C 180,E1 -14127.629,E2 -14127.629} C_VEL
LIN {X 0,Y 339.656,Z 619.121,A -85,B 0,C 180,E1 -14128.816,E2 -14128.816} C_VEL
LIN {X 0,Y 339.629,Z 619.853,A -85,B 0,C 180,E1 -14130.001,E2 -14130.001} C_VEL
LIN {X 0,Y 339.464,Z 620.087,A -85,B 0,C 180,E1 -14131.188,E2 -14131.188} C_VEL
LIN {X 0,Y 339.431,Z 619.899,A -85,B 0,C 180,E1 -14132.375,E2 -14132.375} C_VEL
LIN {X 0,Y 339.252,Z 619.267,A -85,B 0,C 180,E1 -14133.564,E2 -14133.564} C_VEL
LIN {X 0,Y 339.241,Z 618.169,A -85,B 0,C 180,E1 -14134.755,E2 -14134.755} C_VEL
LIN {X 0,Y 339.254,Z 616.426,A -85,B 0,C 180,E1 -14136.081,E2 -14136.081} C_VEL
LIN {X 0,Y 339.35,Z 613.461,A -85,B 0,C 180,E1 -14137.738,E2 -14137.738} C_VEL
LIN {X 0,Y 339.651,Z 609.208,A -85,B 0,C 180,E1 -14139.53,E2 -14139.53} C_VEL
LIN {X 0,Y 340.343,Z 602.785,A -85,B 0,C 180,E1 -14141.616,E2 -14141.616} C_VEL
LIN {X 0,Y 341.281,Z 595.808,A -85,B 0,C 180,E1 -14143.397,E2 -14143.397} C_VEL
LIN {X 0,Y 342.559,Z 587.129,A -85,B 0,C 180,E1 -14145.183,E2 -14145.183} C_VEL
LIN {X 0,Y 343.919,Z 578.6,A -85,B 0,C 180,E1 -14146.625,E2 -14146.625} C_VEL
LIN {X 0,Y 345.627,Z 568.234,A -85,B 0,C 180,E1 -14148.066,E2 -14148.066} C_VEL
LIN {X 0,Y 347.603,Z 555.405,A -85,B 0,C 180,E1 -14149.489,E2 -14149.489} C_VEL
LIN {X 0,Y 349.379,Z 542.465,A -85,B 0,C 180,E1 -14150.612,E2 -14150.612} C_VEL
LIN {X 0,Y 351.259,Z 528.878,A -85,B 0,C 180,E1 -14151.495,E2 -14151.495} C_VEL
LIN {X 0,Y 352.732,Z 514.554,A -85,B 0,C 180,E1 -14152.169,E2 -14152.169} C_VEL
LIN {X 0,Y 356.644,Z 450.728,A -85,B 0,C 180,E1 -14154.287,E2 -14154.287} C_VEL
LIN {X 0,Y 355.528,Z 435.935,A -85,B 0,C 180,E1 -14155.064,E2 -14155.064} C_VEL
LIN {X 0,Y 353.392,Z 421.489,A -85,B 0,C 180,E1 -14156.011,E2 -14156.011} C_VEL
LIN {X 0,Y 350.253,Z 406.438,A -85,B 0,C 180,E1 -14157.214,E2 -14157.214} C_VEL
LIN {X 0,Y 348.641,Z 399.319,A -85,B 0,C 180,E1 -14157.843,E2 -14157.843} C_VEL
LIN {X 0,Y 349.172,Z 396.607,A -85,B 0,C 180,E1 -14158.558,E2 -14158.558} C_VEL
LIN {X 0,Y 347.911,Z 389.206,A -85,B 0,C 180,E1 -14161.006,E2 -14161.006} C_VEL
LIN {X 0,Y 346.147,Z 381.499,A -85,B 0,C 180,E1 -14164.004,E2 -14164.004} C_VEL
LIN {X 0,Y 344.833,Z 376.697,A -85,B 0,C 180,E1 -14166.233,E2 -14166.233} C_VEL
LIN {X 0,Y 343.058,Z 371.22,A -85,B 0,C 180,E1 -14169.427,E2 -14169.427} C_VEL
LIN {X 0,Y 341.746,Z 367.123,A -85,B 0,C 180,E1 -14172.739,E2 -14172.739} C_VEL
LIN {X 0,Y 340.753,Z 364.572,A -85,B 0,C 180,E1 -14176.211,E2 -14176.211} C_VEL
LIN {X 0,Y 340.704,Z 364.044,A -85,B 0,C 180,E1 -14177.955,E2 -14177.955} C_VEL
LIN {X 0,Y 340.739,Z 364.043,A -85,B 0,C 180,E1 -14181.773,E2 -14181.773} C_VEL
LIN {X 0,Y 340.809,Z 364.559,A -85,B 0,C 180,E1 -14183.539,E2 -14183.539} C_VEL
LIN {X 0,Y 341.378,Z 366.261,A -85,B 0,C 180,E1 -14186.23,E2 -14186.23} C_VEL
LIN {X 0,Y 342.403,Z 369.59,A -85,B 0,C 180,E1 -14189.552,E2 -14189.552} C_VEL
LIN {X 0,Y 343.147,Z 371.885,A -85,B 0,C 180,E1 -14191.216,E2 -14191.216} C_VEL
LIN {X 0,Y 345.651,Z 375.416,A -85,B 0,C 180,E1 -14191.944,E2 -14191.944} C_VEL
LIN {X 0,Y 349.746,Z 381.353,A -85,B 0,C 180,E1 -14193.048,E2 -14193.048} C_VEL
LIN {X 0,Y 355.043,Z 389.94,A -85,B 0,C 180,E1 -14194.37,E2 -14194.37} C_VEL
LIN {X 0,Y 359.393,Z 398.42,A -85,B 0,C 180,E1 -14195.414,E2 -14195.414} C_VEL
LIN {X 0,Y 354.247,Z 472.359,A -85,B 0,C 180,E1 -14197.894,E2 -14197.894} C_VEL
LIN {X 0,Y 353.299,Z 485.869,A -85,B 0,C 180,E1 -14198.56,E2 -14198.56} C_VEL
LIN {X 0,Y 352.186,Z 498.396,A -85,B 0,C 180,E1 -14199.408,E2 -14199.408} C_VEL
LIN {X 0,Y 350.768,Z 510.614,A -85,B 0,C 180,E1 -14200.484,E2 -14200.484} C_VEL
LIN {X 0,Y 349.119,Z 522.527,A -85,B 0,C 180,E1 -14201.819,E2 -14201.819} C_VEL
LIN {X 0,Y 347.444,Z 532.726,A -85,B 0,C 180,E1 -14203.247,E2 -14203.247} C_VEL
LIN {X 0,Y 346.015,Z 541.084,A -85,B 0,C 180,E1 -14204.69,E2 -14204.69} C_VEL
LIN {X 0,Y 344.574,Z 549.215,A -85,B 0,C 180,E1 -14206.434,E2 -14206.434} C_VEL
LIN {X 0,Y 343.283,Z 555.758,A -85,B 0,C 180,E1 -14208.186,E2 -14208.186} C_VEL
LIN {X 0,Y 342.269,Z 560.937,A -85,B 0,C 180,E1 -14209.948,E2 -14209.948} C_VEL
LIN {X 0,Y 341.255,Z 564.956,A -85,B 0,C 180,E1 -14211.711,E2 -14211.711} C_VEL
LIN {X 0,Y 340.903,Z 567.005,A -85,B 0,C 180,E1 -14212.894,E2 -14212.894} C_VEL
LIN {X 0,Y 340.547,Z 568.567,A -85,B 0,C 180,E1 -14214.077,E2 -14214.077} C_VEL
LIN {X 0,Y 340.429,Z 569.691,A -85,B 0,C 180,E1 -14215.263,E2 -14215.263} C_VEL
LIN {X 0,Y 340.163,Z 570.427,A -85,B 0,C 180,E1 -14216.446,E2 -14216.446} C_VEL
LIN {X 0,Y 339.864,Z 570.698,A -85,B 0,C 180,E1 -14217.63,E2 -14217.63} C_VEL
LIN {X 0,Y 339.615,Z 570.547,A -85,B 0,C 180,E1 -14218.814,E2 -14218.814} C_VEL
LIN {X 0,Y 339.504,Z 569.975,A -85,B 0,C 180,E1 -14220,E2 -14220} C_VEL
LIN {X 0,Y 339.494,Z 568.949,A -85,B 0,C 180,E1 -14221.186,E2 -14221.186} C_VEL
LIN {X 0,Y 339.568,Z 567.467,A -85,B 0,C 180,E1 -14222.372,E2 -14222.372} C_VEL
LIN {X 0,Y 339.66,Z 564.414,A -85,B 0,C 180,E1 -14224.153,E2 -14224.153} C_VEL
LIN {X 0,Y 339.866,Z 559.311,A -85,B 0,C 180,E1 -14226.293,E2 -14226.293} C_VEL
LIN {X 0,Y 340.182,Z 552.796,A -85,B 0,C 180,E1 -14228.315,E2 -14228.315} C_VEL
LIN {X 0,Y 340.696,Z 545.523,A -85,B 0,C 180,E1 -14230.098,E2 -14230.098} C_VEL
LIN {X 0,Y 341.232,Z 538.109,A -85,B 0,C 180,E1 -14231.584,E2 -14231.584} C_VEL
LIN {X 0,Y 341.945,Z 528.136,A -85,B 0,C 180,E1 -14233.218,E2 -14233.218} C_VEL
LIN {X 0,Y 342.706,Z 516.925,A -85,B 0,C 180,E1 -14234.701,E2 -14234.701} C_VEL
LIN {X 0,Y 343.384,Z 506.048,A -85,B 0,C 180,E1 -14235.855,E2 -14235.855} C_VEL
LIN {X 0,Y 344.094,Z 493.384,A -85,B 0,C 180,E1 -14236.921,E2 -14236.921} C_VEL
LIN {X 0,Y 344.678,Z 480.699,A -85,B 0,C 180,E1 -14237.733,E2 -14237.733} C_VEL
LIN {X 0,Y 345.114,Z 466.864,A -85,B 0,C 180,E1 -14238.361,E2 -14238.361} C_VEL
LIN {X 0,Y 347.335,Z 384.206,A -85,B 0,C 180,E1 -14240.709,E2 -14240.709} C_VEL
LIN {X 0,Y 340.772,Z 364.034,A -85,B 0,C 180,E1 -14241.592,E2 -14241.592} C_VEL
LIN {X 0,Y 340.778,Z 364.034,A -85,B 0,C 180,E1 -14245.664,E2 -14245.664} C_VEL
LIN {X 0,Y 340.746,Z 364.042,A -85,B 0,C 180,E1 -14248.319,E2 -14248.319} C_VEL
LIN {X 0,Y 340.709,Z 364.043,A -85,B 0,C 180,E1 -14251.043,E2 -14251.043} C_VEL
LIN {X 0,Y 340.723,Z 364.04,A -85,B 0,C 180,E1 -14255.278,E2 -14255.278} C_VEL
LIN {X 0,Y 340.715,Z 364.046,A -85,B 0,C 180,E1 -14258.385,E2 -14258.385} C_VEL
LIN {X 0,Y 340.703,Z 364.047,A -85,B 0,C 180,E1 -14262.045,E2 -14262.045} C_VEL
LIN {X 0,Y 340.656,Z 364.054,A -85,B 0,C 180,E1 -14266.226,E2 -14266.226} C_VEL
LIN {X 0,Y 340.692,Z 364.046,A -85,B 0,C 180,E1 -14269.752,E2 -14269.752} C_VEL
LIN {X 0,Y 340.709,Z 364.042,A -85,B 0,C 180,E1 -14273.258,E2 -14273.258} C_VEL
LIN {X 0,Y 340.698,Z 364.048,A -85,B 0,C 180,E1 -14276.153,E2 -14276.153} C_VEL
LIN {X 0,Y 340.745,Z 364.042,A -85,B 0,C 180,E1 -14280.328,E2 -14280.328} C_VEL
LIN {X 0,Y 340.808,Z 364.03,A -85,B 0,C 180,E1 -14283.019,E2 -14283.019} C_VEL
LIN {X 0,Y 340.732,Z 364.039,A -85,B 0,C 180,E1 -14286.926,E2 -14286.926} C_VEL
LIN {X 0,Y 340.798,Z 364.032,A -85,B 0,C 180,E1 -14290.733,E2 -14290.733} C_VEL
LIN {X 0,Y 340.79,Z 364.032,A -85,B 0,C 180,E1 -14293.218,E2 -14293.218} C_VEL
LIN {X 0,Y 340.847,Z 364.025,A -85,B 0,C 180,E1 -14296.889,E2 -14296.889} C_VEL
LIN {X 0,Y 340.916,Z 364.018,A -85,B 0,C 180,E1 -14300.506,E2 -14300.506} C_VEL
LIN {X 0,Y 341.061,Z 363.998,A -85,B 0,C 180,E1 -14302.897,E2 -14302.897} C_VEL
LIN {X 0,Y 341.172,Z 363.987,A -85,B 0,C 180,E1 -14307.637,E2 -14307.637} C_VEL
LIN {X 0,Y 341.318,Z 363.971,A -85,B 0,C 180,E1 -14309.999,E2 -14309.999} C_VEL
LIN {X 0,Y 341.172,Z 363.987,A -85,B 0,C 180,E1 -14312.36,E2 -14312.36} C_VEL
LIN {X 0,Y 341.077,Z 363.996,A -85,B 0,C 180,E1 -14317.1,E2 -14317.1} C_VEL
LIN {X 0,Y 340.871,Z 364.022,A -85,B 0,C 180,E1 -14320.692,E2 -14320.692} C_VEL
LIN {X 0,Y 340.862,Z 364.025,A -85,B 0,C 180,E1 -14324.323,E2 -14324.323} C_VEL
LIN {X 0,Y 340.836,Z 364.027,A -85,B 0,C 180,E1 -14328.466,E2 -14328.466} C_VEL
LIN {X 0,Y 340.751,Z 364.042,A -85,B 0,C 180,E1 -14331.855,E2 -14331.855} C_VEL
LIN {X 0,Y 340.769,Z 364.038,A -85,B 0,C 180,E1 -14335.663,E2 -14335.663} C_VEL
LIN {X 0,Y 340.738,Z 364.04,A -85,B 0,C 180,E1 -14338.318,E2 -14338.318} C_VEL
LIN {X 0,Y 340.712,Z 364.042,A -85,B 0,C 180,E1 -14341.041,E2 -14341.041} C_VEL
LIN {X 0,Y 340.714,Z 364.043,A -85,B 0,C 180,E1 -14345.277,E2 -14345.277} C_VEL
LIN {X 0,Y 340.714,Z 364.042,A -85,B 0,C 180,E1 -14348.387,E2 -14348.387} C_VEL
LIN {X 0,Y 340.719,Z 364.042,A -85,B 0,C 180,E1 -14351.302,E2 -14351.302} C_VEL
LIN {X 0,Y 340.775,Z 364.034,A -85,B 0,C 180,E1 -14354.521,E2 -14354.521} C_VEL
LIN {X 0,Y 340.747,Z 364.041,A -85,B 0,C 180,E1 -14357.943,E2 -14357.943} C_VEL
LIN {X 0,Y 340.741,Z 364.041,A -85,B 0,C 180,E1 -14359.535,E2 -14359.535} C_VEL
LIN {X 0,Y 340.115,Z 364.126,A -85,B 0,C 180,E1 -14360.521,E2 -14360.521} C_VEL
LIN {X 0,Y 337.232,Z 364.484,A -85,B 0,C 180,E1 -14362.125,E2 -14362.125} C_VEL
LIN {X 0,Y 334.77,Z 364.785,A -85,B 0,C 180,E1 -14363.424,E2 -14363.424} C_VEL
LIN {X 0,Y 333.728,Z 364.912,A -85,B 0,C 180,E1 -14364.43,E2 -14364.43} C_VEL
LIN {X 0,Y 333.653,Z 364.92,A -85,B 0,C 180,E1 -14364.771,E2 -14364.771} C_VEL
LIN {X 0,Y 333.625,Z 364.925,A -85,B 0,C 180,E1 -14368.221,E2 -14368.221} C_VEL
LIN {X 0,Y 333.703,Z 364.915,A -85,B 0,C 180,E1 -14371.027,E2 -14371.027} C_VEL
LIN {X 0,Y 333.727,Z 364.916,A -85,B 0,C 180,E1 -14373.753,E2 -14373.753} C_VEL
LIN {X 0,Y 333.71,Z 364.916,A -85,B 0,C 180,E1 -14377.913,E2 -14377.913} C_VEL
LIN {X 0,Y 333.785,Z 364.91,A -85,B 0,C 180,E1 -14381.589,E2 -14381.589} C_VEL
LIN {X 0,Y 333.799,Z 364.908,A -85,B 0,C 180,E1 -14385.576,E2 -14385.576} C_VEL
LIN {X 0,Y 333.828,Z 364.9,A -85,B 0,C 180,E1 -14389.078,E2 -14389.078} C_VEL
LIN {X 0,Y 334.016,Z 364.875,A -85,B 0,C 180,E1 -14392.747,E2 -14392.747} C_VEL
LIN {X 0,Y 333.804,Z 364.904,A -85,B 0,C 180,E1 -14395.169,E2 -14395.169} C_VEL
LIN {X 0,Y 334.122,Z 364.867,A -85,B 0,C 180,E1 -14397.589,E2 -14397.589} C_VEL
LIN {X 0,Y 334.258,Z 364.846,A -85,B 0,C 180,E1 -14400,E2 -14400} C_VEL
LIN {X 0,Y 334.099,Z 364.865,A -85,B 0,C 180,E1 -14402.411,E2 -14402.411} C_VEL
LIN {X 0,Y 334.015,Z 364.876,A -85,B 0,C 180,E1 -14406.039,E2 -14406.039} C_VEL
LIN {X 0,Y 333.975,Z 364.88,A -85,B 0,C 180,E1 -14408.502,E2 -14408.502} C_VEL
LIN {X 0,Y 333.787,Z 364.904,A -85,B 0,C 180,E1 -14412.155,E2 -14412.155} C_VEL
LIN {X 0,Y 333.769,Z 364.908,A -85,B 0,C 180,E1 -14415.887,E2 -14415.887} C_VEL
LIN {X 0,Y 333.787,Z 364.904,A -85,B 0,C 180,E1 -14418.656,E2 -14418.656} C_VEL
LIN {X 0,Y 333.684,Z 364.917,A -85,B 0,C 180,E1 -14422.279,E2 -14422.279} C_VEL
LIN {X 0,Y 333.727,Z 364.911,A -85,B 0,C 180,E1 -14426.247,E2 -14426.247} C_VEL
LIN {X 0,Y 333.682,Z 364.919,A -85,B 0,C 180,E1 -14428.975,E2 -14428.975} C_VEL
LIN {X 0,Y 333.636,Z 364.923,A -85,B 0,C 180,E1 -14432.588,E2 -14432.588} C_VEL
LIN {X 0,Y 333.671,Z 364.918,A -85,B 0,C 180,E1 -14436.14,E2 -14436.14} C_VEL
LIN {X 0,Y 333.681,Z 364.922,A -85,B 0,C 180,E1 -14439.188,E2 -14439.188} C_VEL
LIN {X 0,Y 333.697,Z 364.915,A -85,B 0,C 180,E1 -14442.515,E2 -14442.515} C_VEL
LIN {X 0,Y 333.723,Z 364.912,A -85,B 0,C 180,E1 -14445.978,E2 -14445.978} C_VEL
LIN {X 0,Y 333.697,Z 364.92,A -85,B 0,C 180,E1 -14449.306,E2 -14449.306} C_VEL
LIN {X 0,Y 333.662,Z 364.925,A -85,B 0,C 180,E1 -14453.169,E2 -14453.169} C_VEL
LIN {X 0,Y 333.651,Z 364.923,A -85,B 0,C 180,E1 -14456.795,E2 -14456.795} C_VEL
LIN {X 0,Y 333.733,Z 365.117,A -85,B 0,C 180,E1 -14457.806,E2 -14457.806} C_VEL
LIN {X 0,Y 336.69,Z 379.495,A -85,B 0,C 180,E1 -14461.31,E2 -14461.31} C_VEL
LIN {X 0,Y 337.896,Z 385.679,A -85,B 0,C 180,E1 -14462.77,E2 -14462.77} C_VEL
LIN {X 0,Y 336.993,Z 395.844,A -85,B 0,C 180,E1 -14465.021,E2 -14465.021} C_VEL
LIN {X 0,Y 335.692,Z 408.925,A -85,B 0,C 180,E1 -14467.892,E2 -14467.892} C_VEL
LIN {X 0,Y 338.662,Z 439.866,A -85,B 0,C 180,E1 -14468.967,E2 -14468.967} C_VEL
LIN {X 0,Y 339.729,Z 449.785,A -85,B 0,C 180,E1 -14469.309,E2 -14469.309} C_VEL
LIN {X 0,Y 337.86,Z 519.536,A -85,B 0,C 180,E1 -14471.389,E2 -14471.389} C_VEL
LIN {X 0,Y 337.073,Z 532.746,A -85,B 0,C 180,E1 -14472.012,E2 -14472.012} C_VEL
LIN {X 0,Y 336.248,Z 545.088,A -85,B 0,C 180,E1 -14472.83,E2 -14472.83} C_VEL
LIN {X 0,Y 335.455,Z 557.206,A -85,B 0,C 180,E1 -14473.885,E2 -14473.885} C_VEL
LIN {X 0,Y 334.743,Z 567.194,A -85,B 0,C 180,E1 -14474.969,E2 -14474.969} C_VEL
LIN {X 0,Y 334.027,Z 577.311,A -85,B 0,C 180,E1 -14476.31,E2 -14476.31} C_VEL
LIN {X 0,Y 333.379,Z 586.638,A -85,B 0,C 180,E1 -14477.832,E2 -14477.832} C_VEL
LIN {X 0,Y 332.789,Z 595.737,A -85,B 0,C 180,E1 -14479.66,E2 -14479.66} C_VEL
LIN {X 0,Y 332.521,Z 602.963,A -85,B 0,C 180,E1 -14481.493,E2 -14481.493} C_VEL
LIN {X 0,Y 332.41,Z 609.353,A -85,B 0,C 180,E1 -14483.568,E2 -14483.568} C_VEL
LIN {X 0,Y 332.354,Z 613.064,A -85,B 0,C 180,E1 -14485.149,E2 -14485.149} C_VEL
LIN {X 0,Y 332.421,Z 615.346,A -85,B 0,C 180,E1 -14486.365,E2 -14486.365} C_VEL
LIN {X 0,Y 332.461,Z 617.077,A -85,B 0,C 180,E1 -14487.578,E2 -14487.578} C_VEL
LIN {X 0,Y 332.609,Z 618.351,A -85,B 0,C 180,E1 -14488.791,E2 -14488.791} C_VEL
LIN {X 0,Y 332.583,Z 619.162,A -85,B 0,C 180,E1 -14490.001,E2 -14490.001} C_VEL
LIN {X 0,Y 332.398,Z 619.475,A -85,B 0,C 180,E1 -14491.213,E2 -14491.213} C_VEL
LIN {X 0,Y 332.347,Z 619.335,A -85,B 0,C 180,E1 -14492.425,E2 -14492.425} C_VEL
LIN {X 0,Y 332.169,Z 618.755,A -85,B 0,C 180,E1 -14493.641,E2 -14493.641} C_VEL
LIN {X 0,Y 332.155,Z 617.754,A -85,B 0,C 180,E1 -14494.856,E2 -14494.856} C_VEL
LIN {X 0,Y 332.182,Z 616.267,A -85,B 0,C 180,E1 -14496.074,E2 -14496.074} C_VEL
LIN {X 0,Y 332.267,Z 613.219,A -85,B 0,C 180,E1 -14497.904,E2 -14497.904} C_VEL
LIN {X 0,Y 332.614,Z 609.09,A -85,B 0,C 180,E1 -14499.733,E2 -14499.733} C_VEL
LIN {X 0,Y 333.377,Z 602.807,A -85,B 0,C 180,E1 -14501.863,E2 -14501.863} C_VEL
LIN {X 0,Y 334.366,Z 596.018,A -85,B 0,C 180,E1 -14503.679,E2 -14503.679} C_VEL
LIN {X 0,Y 335.647,Z 588.039,A -85,B 0,C 180,E1 -14505.414,E2 -14505.414} C_VEL
LIN {X 0,Y 337.172,Z 579.281,A -85,B 0,C 180,E1 -14506.968,E2 -14506.968} C_VEL
LIN {X 0,Y 339.153,Z 568.114,A -85,B 0,C 180,E1 -14508.58,E2 -14508.58} C_VEL
LIN {X 0,Y 341.021,Z 556.916,A -85,B 0,C 180,E1 -14509.881,E2 -14509.881} C_VEL
LIN {X 0,Y 342.896,Z 544.638,A -85,B 0,C 180,E1 -14511.02,E2 -14511.02} C_VEL
LIN {X 0,Y 344.781,Z 532.048,A -85,B 0,C 180,E1 -14511.919,E2 -14511.919} C_VEL
LIN {X 0,Y 346.565,Z 517.188,A -85,B 0,C 180,E1 -14512.703,E2 -14512.703} C_VEL
LIN {X 0,Y 347.947,Z 497.154,A -85,B 0,C 180,E1 -14513.433,E2 -14513.433} C_VEL
LIN {X 0,Y 351.052,Z 452.59,A -85,B 0,C 180,E1 -14514.933,E2 -14514.933} C_VEL
LIN {X 0,Y 350.15,Z 438.338,A -85,B 0,C 180,E1 -14515.702,E2 -14515.702} C_VEL
LIN {X 0,Y 348.144,Z 423.956,A -85,B 0,C 180,E1 -14516.688,E2 -14516.688} C_VEL
LIN {X 0,Y 345.407,Z 409.821,A -85,B 0,C 180,E1 -14517.857,E2 -14517.857} C_VEL
LIN {X 0,Y 343.145,Z 400.308,A -85,B 0,C 180,E1 -14518.782,E2 -14518.782} C_VEL
LIN {X 0,Y 342.508,Z 398.056,A -85,B 0,C 180,E1 -14519.065,E2 -14519.065} C_VEL
LIN {X 0,Y 341.287,Z 391.267,A -85,B 0,C 180,E1 -14521.44,E2 -14521.44} C_VEL
LIN {X 0,Y 339.488,Z 383.328,A -85,B 0,C 180,E1 -14524.702,E2 -14524.702} C_VEL
LIN {X 0,Y 338.139,Z 378.674,A -85,B 0,C 180,E1 -14527.068,E2 -14527.068} C_VEL
LIN {X 0,Y 336.933,Z 374.748,A -85,B 0,C 180,E1 -14529.486,E2 -14529.486} C_VEL
LIN {X 0,Y 335.637,Z 370.683,A -85,B 0,C 180,E1 -14532.872,E2 -14532.872} C_VEL
LIN {X 0,Y 334.733,Z 368.342,A -85,B 0,C 180,E1 -14536.143,E2 -14536.143} C_VEL
LIN {X 0,Y 334.596,Z 367.644,A -85,B 0,C 180,E1 -14537.767,E2 -14537.767} C_VEL
LIN {X 0,Y 334.461,Z 367.437,A -85,B 0,C 180,E1 -14541.032,E2 -14541.032} C_VEL
LIN {X 0,Y 334.663,Z 367.892,A -85,B 0,C 180,E1 -14542.942,E2 -14542.942} C_VEL
LIN {X 0,Y 335.01,Z 369.319,A -85,B 0,C 180,E1 -14545.499,E2 -14545.499} C_VEL
LIN {X 0,Y 335.769,Z 371.829,A -85,B 0,C 180,E1 -14548.447,E2 -14548.447} C_VEL
LIN {X 0,Y 336.315,Z 373.375,A -85,B 0,C 180,E1 -14549.734,E2 -14549.734} C_VEL
LIN {X 0,Y 338.991,Z 376.999,A -85,B 0,C 180,E1 -14550.618,E2 -14550.618} C_VEL
LIN {X 0,Y 340.488,Z 379.016,A -85,B 0,C 180,E1 -14551.08,E2 -14551.08} C_VEL
LIN {X 0,Y 343.227,Z 382.747,A -85,B 0,C 180,E1 -14551.883,E2 -14551.883} C_VEL
LIN {X 0,Y 347.652,Z 389.54,A -85,B 0,C 180,E1 -14553.111,E2 -14553.111} C_VEL
LIN {X 0,Y 352.734,Z 398.637,A -85,B 0,C 180,E1 -14554.43,E2 -14554.43} C_VEL
LIN {X 0,Y 353.945,Z 401.168,A -85,B 0,C 180,E1 -14554.742,E2 -14554.742} C_VEL
LIN {X 0,Y 348.492,Z 473.232,A -85,B 0,C 180,E1 -14557.235,E2 -14557.235} C_VEL
LIN {X 0,Y 347.41,Z 487.159,A -85,B 0,C 180,E1 -14557.944,E2 -14557.944} C_VEL
LIN {X 0,Y 346.304,Z 498.694,A -85,B 0,C 180,E1 -14558.746,E2 -14558.746} C_VEL
LIN {X 0,Y 344.931,Z 509.91,A -85,B 0,C 180,E1 -14559.734,E2 -14559.734} C_VEL
LIN {X 0,Y 343.198,Z 521.614,A -85,B 0,C 180,E1 -14561.029,E2 -14561.029} C_VEL
LIN {X 0,Y 341.567,Z 531.151,A -85,B 0,C 180,E1 -14562.332,E2 -14562.332} C_VEL
LIN {X 0,Y 339.674,Z 541.397,A -85,B 0,C 180,E1 -14564.089,E2 -14564.089} C_VEL
LIN {X 0,Y 338.09,Z 549.599,A -85,B 0,C 180,E1 -14565.862,E2 -14565.862} C_VEL
LIN {X 0,Y 336.492,Z 557.148,A -85,B 0,C 180,E1 -14567.944,E2 -14567.944} C_VEL
LIN {X 0,Y 335.395,Z 562.164,A -85,B 0,C 180,E1 -14569.74,E2 -14569.74} C_VEL
LIN {X 0,Y 334.317,Z 566.037,A -85,B 0,C 180,E1 -14571.538,E2 -14571.538} C_VEL
LIN {X 0,Y 333.924,Z 567.958,A -85,B 0,C 180,E1 -14572.745,E2 -14572.745} C_VEL
LIN {X 0,Y 333.542,Z 569.449,A -85,B 0,C 180,E1 -14573.952,E2 -14573.952} C_VEL
LIN {X 0,Y 333.411,Z 570.507,A -85,B 0,C 180,E1 -14575.163,E2 -14575.163} C_VEL
LIN {X 0,Y 333.137,Z 571.126,A -85,B 0,C 180,E1 -14576.371,E2 -14576.371} C_VEL
LIN {X 0,Y 332.798,Z 571.324,A -85,B 0,C 180,E1 -14577.579,E2 -14577.579} C_VEL
LIN {X 0,Y 332.547,Z 571.105,A -85,B 0,C 180,E1 -14578.789,E2 -14578.789} C_VEL
LIN {X 0,Y 332.436,Z 570.447,A -85,B 0,C 180,E1 -14580,E2 -14580} C_VEL
LIN {X 0,Y 332.43,Z 569.319,A -85,B 0,C 180,E1 -14581.211,E2 -14581.211} C_VEL
LIN {X 0,Y 332.492,Z 567.769,A -85,B 0,C 180,E1 -14582.423,E2 -14582.423} C_VEL
LIN {X 0,Y 332.577,Z 564.585,A -85,B 0,C 180,E1 -14584.241,E2 -14584.241} C_VEL
LIN {X 0,Y 332.753,Z 560.291,A -85,B 0,C 180,E1 -14586.062,E2 -14586.062} C_VEL
LIN {X 0,Y 333.048,Z 554.762,A -85,B 0,C 180,E1 -14587.884,E2 -14587.884} C_VEL
LIN {X 0,Y 333.459,Z 547.779,A -85,B 0,C 180,E1 -14589.707,E2 -14589.707} C_VEL
LIN {X 0,Y 334.096,Z 539.113,A -85,B 0,C 180,E1 -14591.528,E2 -14591.528} C_VEL
LIN {X 0,Y 334.825,Z 529.266,A -85,B 0,C 180,E1 -14593.195,E2 -14593.195} C_VEL
LIN {X 0,Y 335.588,Z 518.17,A -85,B 0,C 180,E1 -14594.71,E2 -14594.71} C_VEL
LIN {X 0,Y 336.308,Z 507.354,A -85,B 0,C 180,E1 -14595.903,E2 -14595.903} C_VEL
LIN {X 0,Y 336.923,Z 495.077,A -85,B 0,C 180,E1 -14596.979,E2 -14596.979} C_VEL
LIN {X 0,Y 337.587,Z 482.874,A -85,B 0,C 180,E1 -14597.804,E2 -14597.804} C_VEL
LIN {X 0,Y 338.072,Z 468.878,A -85,B 0,C 180,E1 -14598.483,E2 -14598.483} C_VEL
LIN {X 0,Y 338.926,Z 435.609,A -85,B 0,C 180,E1 -14599.485,E2 -14599.485} C_VEL
LIN {X 0,Y 340.309,Z 385.364,A -85,B 0,C 180,E1 -14600.949,E2 -14600.949} C_VEL
LIN {X 0,Y 333.715,Z 364.915,A -85,B 0,C 180,E1 -14601.862,E2 -14601.862} C_VEL
LIN {X 0,Y 333.724,Z 364.912,A -85,B 0,C 180,E1 -14605.1,E2 -14605.1} C_VEL
LIN {X 0,Y 333.725,Z 364.913,A -85,B 0,C 180,E1 -14607.809,E2 -14607.809} C_VEL
LIN {X 0,Y 333.702,Z 364.92,A -85,B 0,C 180,E1 -14610.362,E2 -14610.362} C_VEL
LIN {X 0,Y 333.69,Z 364.918,A -85,B 0,C 180,E1 -14614.773,E2 -14614.773} C_VEL
LIN {X 0,Y 333.657,Z 364.921,A -85,B 0,C 180,E1 -14617.65,E2 -14617.65} C_VEL
LIN {X 0,Y 333.651,Z 364.923,A -85,B 0,C 180,E1 -14620.767,E2 -14620.767} C_VEL
LIN {X 0,Y 333.598,Z 364.933,A -85,B 0,C 180,E1 -14624.25,E2 -14624.25} C_VEL
LIN {X 0,Y 333.646,Z 364.923,A -85,B 0,C 180,E1 -14627.618,E2 -14627.618} C_VEL
LIN {X 0,Y 333.657,Z 364.92,A -85,B 0,C 180,E1 -14631.201,E2 -14631.201} C_VEL
LIN {X 0,Y 333.68,Z 364.92,A -85,B 0,C 180,E1 -14633.86,E2 -14633.86} C_VEL
LIN {X 0,Y 333.649,Z 364.921,A -85,B 0,C 180,E1 -14637.411,E2 -14637.411} C_VEL
LIN {X 0,Y 333.694,Z 364.916,A -85,B 0,C 180,E1 -14641.025,E2 -14641.025} C_VEL
LIN {X 0,Y 333.739,Z 364.912,A -85,B 0,C 180,E1 -14643.753,E2 -14643.753} C_VEL
LIN {X 0,Y 333.723,Z 364.916,A -85,B 0,C 180,E1 -14647.913,E2 -14647.913} C_VEL
LIN {X 0,Y 333.798,Z 364.904,A -85,B 0,C 180,E1 -14651.588,E2 -14651.588} C_VEL
LIN {X 0,Y 333.811,Z 364.903,A -85,B 0,C 180,E1 -14655.575,E2 -14655.575} C_VEL
LIN {X 0,Y 333.837,Z 364.898,A -85,B 0,C 180,E1 -14659.077,E2 -14659.077} C_VEL
LIN {X 0,Y 334.008,Z 364.877,A -85,B 0,C 180,E1 -14662.746,E2 -14662.746} C_VEL
LIN {X 0,Y 333.812,Z 364.901,A -85,B 0,C 180,E1 -14665.168,E2 -14665.168} C_VEL
LIN {X 0,Y 334.109,Z 364.866,A -85,B 0,C 180,E1 -14667.587,E2 -14667.587} C_VEL
LIN {X 0,Y 334.268,Z 364.85,A -85,B 0,C 180,E1 -14669.999,E2 -14669.999} C_VEL
LIN {X 0,Y 334.109,Z 364.866,A -85,B 0,C 180,E1 -14672.41,E2 -14672.41} C_VEL
LIN {X 0,Y 334.026,Z 364.875,A -85,B 0,C 180,E1 -14677.251,E2 -14677.251} C_VEL
LIN {X 0,Y 333.834,Z 364.898,A -85,B 0,C 180,E1 -14680.92,E2 -14680.92} C_VEL
LIN {X 0,Y 333.807,Z 364.902,A -85,B 0,C 180,E1 -14684.633,E2 -14684.633} C_VEL
LIN {X 0,Y 333.795,Z 364.903,A -85,B 0,C 180,E1 -14688.654,E2 -14688.654} C_VEL
LIN {X 0,Y 333.69,Z 364.918,A -85,B 0,C 180,E1 -14692.277,E2 -14692.277} C_VEL
LIN {X 0,Y 333.733,Z 364.913,A -85,B 0,C 180,E1 -14696.245,E2 -14696.245} C_VEL
LIN {X 0,Y 333.708,Z 364.914,A -85,B 0,C 180,E1 -14698.97,E2 -14698.97} C_VEL
LIN {X 0,Y 333.647,Z 364.922,A -85,B 0,C 180,E1 -14702.588,E2 -14702.588} C_VEL
LIN {X 0,Y 333.672,Z 364.921,A -85,B 0,C 180,E1 -14706.137,E2 -14706.137} C_VEL
LIN {X 0,Y 333.679,Z 364.918,A -85,B 0,C 180,E1 -14709.186,E2 -14709.186} C_VEL
LIN {X 0,Y 333.697,Z 364.915,A -85,B 0,C 180,E1 -14712.512,E2 -14712.512} C_VEL
LIN {X 0,Y 333.723,Z 364.915,A -85,B 0,C 180,E1 -14715.976,E2 -14715.976} C_VEL
LIN {X 0,Y 333.678,Z 364.917,A -85,B 0,C 180,E1 -14719.521,E2 -14719.521} C_VEL
LIN {X 0,Y 333.658,Z 364.921,A -85,B 0,C 180,E1 -14723.166,E2 -14723.166} C_VEL
LIN {X 0,Y 333.653,Z 364.92,A -85,B 0,C 180,E1 -14724.771,E2 -14724.771} C_VEL
LIN {X 0,Y 333.007,Z 365.006,A -85,B 0,C 180,E1 -14725.778,E2 -14725.778} C_VEL
LIN {X 0,Y 330.142,Z 365.361,A -85,B 0,C 180,E1 -14727.415,E2 -14727.415} C_VEL
LIN {X 0,Y 327.719,Z 365.661,A -85,B 0,C 180,E1 -14728.741,E2 -14728.741} C_VEL
LIN {X 0,Y 326.706,Z 365.791,A -85,B 0,C 180,E1 -14729.768,E2 -14729.768} C_VEL
LIN {X 0,Y 326.639,Z 365.794,A -85,B 0,C 180,E1 -14730.116,E2 -14730.116} C_VEL
LIN {X 0,Y 326.677,Z 365.791,A -85,B 0,C 180,E1 -14733.142,E2 -14733.142} C_VEL
LIN {X 0,Y 326.646,Z 365.797,A -85,B 0,C 180,E1 -14735.871,E2 -14735.871} C_VEL
LIN {X 0,Y 326.656,Z 365.795,A -85,B 0,C 180,E1 -14739.865,E2 -14739.865} C_VEL
LIN {X 0,Y 326.691,Z 365.788,A -85,B 0,C 180,E1 -14742.472,E2 -14742.472} C_VEL
LIN {X 0,Y 326.751,Z 365.781,A -85,B 0,C 180,E1 -14746.314,E2 -14746.314} C_VEL
LIN {X 0,Y 326.806,Z 365.775,A -85,B 0,C 180,E1 -14750.094,E2 -14750.094} C_VEL
LIN {X 0,Y 326.97,Z 365.753,A -85,B 0,C 180,E1 -14752.59,E2 -14752.59} C_VEL
LIN {X 0,Y 326.771,Z 365.779,A -85,B 0,C 180,E1 -14755.065,E2 -14755.065} C_VEL
LIN {X 0,Y 327.059,Z 365.748,A -85,B 0,C 180,E1 -14757.537,E2 -14757.537} C_VEL
LIN {X 0,Y 327.209,Z 365.725,A -85,B 0,C 180,E1 -14760,E2 -14760} C_VEL
LIN {X 0,Y 327.04,Z 365.744,A -85,B 0,C 180,E1 -14762.463,E2 -14762.463} C_VEL
LIN {X 0,Y 326.991,Z 365.751,A -85,B 0,C 180,E1 -14766.169,E2 -14766.169} C_VEL
LIN {X 0,Y 326.905,Z 365.761,A -85,B 0,C 180,E1 -14768.655,E2 -14768.655} C_VEL
LIN {X 0,Y 326.73,Z 365.783,A -85,B 0,C 180,E1 -14772.422,E2 -14772.422} C_VEL
LIN {X 0,Y 326.745,Z 365.783,A -85,B 0,C 180,E1 -14774.958,E2 -14774.958} C_VEL
LIN {X 0,Y 326.723,Z 365.785,A -85,B 0,C 180,E1 -14778.839,E2 -14778.839} C_VEL
LIN {X 0,Y 326.612,Z 365.798,A -85,B 0,C 180,E1 -14782.788,E2 -14782.788} C_VEL
LIN {X 0,Y 326.681,Z 365.794,A -85,B 0,C 180,E1 -14785.485,E2 -14785.485} C_VEL
LIN {X 0,Y 326.64,Z 365.797,A -85,B 0,C 180,E1 -14789.661,E2 -14789.661} C_VEL
LIN {X 0,Y 326.6,Z 365.8,A -85,B 0,C 180,E1 -14794.021,E2 -14794.021} C_VEL
LIN {X 0,Y 326.626,Z 365.801,A -85,B 0,C 180,E1 -14797.241,E2 -14797.241} C_VEL
LIN {X 0,Y 326.63,Z 365.795,A -85,B 0,C 180,E1 -14800.204,E2 -14800.204} C_VEL
LIN {X 0,Y 326.652,Z 365.796,A -85,B 0,C 180,E1 -14803.511,E2 -14803.511} C_VEL
LIN {X 0,Y 326.645,Z 365.797,A -85,B 0,C 180,E1 -14807.016,E2 -14807.016} C_VEL
LIN {X 0,Y 326.641,Z 365.796,A -85,B 0,C 180,E1 -14810.767,E2 -14810.767} C_VEL
LIN {X 0,Y 326.609,Z 365.798,A -85,B 0,C 180,E1 -14814.482,E2 -14814.482} C_VEL
LIN {X 0,Y 326.665,Z 365.856,A -85,B 0,C 180,E1 -14817.555,E2 -14817.555} C_VEL
LIN {X 0,Y 329.505,Z 379.605,A -85,B 0,C 180,E1 -14820.985,E2 -14820.985} C_VEL
LIN {X 0,Y 330.877,Z 387.069,A -85,B 0,C 180,E1 -14822.783,E2 -14822.783} C_VEL
LIN {X 0,Y 329.543,Z 400.28,A -85,B 0,C 180,E1 -14825.763,E2 -14825.763} C_VEL
LIN {X 0,Y 328.721,Z 408.668,A -85,B 0,C 180,E1 -14827.617,E2 -14827.617} C_VEL
LIN {X 0,Y 331.549,Z 439.24,A -85,B 0,C 180,E1 -14828.694,E2 -14828.694} C_VEL
LIN {X 0,Y 332.765,Z 449.943,A -85,B 0,C 180,E1 -14829.076,E2 -14829.076} C_VEL
LIN {X 0,Y 330.872,Z 518.462,A -85,B 0,C 180,E1 -14831.182,E2 -14831.182} C_VEL
LIN {X 0,Y 330.061,Z 532.473,A -85,B 0,C 180,E1 -14831.857,E2 -14831.857} C_VEL
LIN {X 0,Y 329.156,Z 545.654,A -85,B 0,C 180,E1 -14832.769,E2 -14832.769} C_VEL
LIN {X 0,Y 328.332,Z 557.533,A -85,B 0,C 180,E1 -14833.845,E2 -14833.845} C_VEL
LIN {X 0,Y 327.507,Z 568.365,A -85,B 0,C 180,E1 -14835.079,E2 -14835.079} C_VEL
LIN {X 0,Y 326.775,Z 579.309,A -85,B 0,C 180,E1 -14836.634,E2 -14836.634} C_VEL
LIN {X 0,Y 326.177,Z 588.227,A -85,B 0,C 180,E1 -14838.19,E2 -14838.19} C_VEL
LIN {X 0,Y 325.646,Z 596.835,A -85,B 0,C 180,E1 -14840.059,E2 -14840.059} C_VEL
LIN {X 0,Y 325.451,Z 603.751,A -85,B 0,C 180,E1 -14841.933,E2 -14841.933} C_VEL
LIN {X 0,Y 325.369,Z 609.188,A -85,B 0,C 180,E1 -14843.801,E2 -14843.801} C_VEL
LIN {X 0,Y 325.317,Z 613.298,A -85,B 0,C 180,E1 -14845.665,E2 -14845.665} C_VEL
LIN {X 0,Y 325.403,Z 616.236,A -85,B 0,C 180,E1 -14847.526,E2 -14847.526} C_VEL
LIN {X 0,Y 325.562,Z 617.569,A -85,B 0,C 180,E1 -14848.764,E2 -14848.764} C_VEL
LIN {X 0,Y 325.537,Z 618.433,A -85,B 0,C 180,E1 -14850.001,E2 -14850.001} C_VEL
LIN {X 0,Y 325.334,Z 618.84,A -85,B 0,C 180,E1 -14851.239,E2 -14851.239} C_VEL
LIN {X 0,Y 325.266,Z 618.773,A -85,B 0,C 180,E1 -14852.478,E2 -14852.478} C_VEL
LIN {X 0,Y 325.088,Z 618.246,A -85,B 0,C 180,E1 -14853.72,E2 -14853.72} C_VEL
LIN {X 0,Y 325.09,Z 616.14,A -85,B 0,C 180,E1 -14856.033,E2 -14856.033} C_VEL
LIN {X 0,Y 325.197,Z 612.992,A -85,B 0,C 180,E1 -14858.077,E2 -14858.077} C_VEL
LIN {X 0,Y 325.568,Z 608.997,A -85,B 0,C 180,E1 -14859.946,E2 -14859.946} C_VEL
LIN {X 0,Y 326.421,Z 602.879,A -85,B 0,C 180,E1 -14862.119,E2 -14862.119} C_VEL
LIN {X 0,Y 327.683,Z 595.041,A -85,B 0,C 180,E1 -14864.281,E2 -14864.281} C_VEL
LIN {X 0,Y 329.196,Z 586.643,A -85,B 0,C 180,E1 -14866.115,E2 -14866.115} C_VEL
LIN {X 0,Y 330.831,Z 578.21,A -85,B 0,C 180,E1 -14867.622,E2 -14867.622} C_VEL
LIN {X 0,Y 332.938,Z 567.018,A -85,B 0,C 180,E1 -14869.26,E2 -14869.26} C_VEL
LIN {X 0,Y 334.951,Z 555.788,A -85,B 0,C 180,E1 -14870.577,E2 -14870.577} C_VEL
LIN {X 0,Y 336.912,Z 543.532,A -85,B 0,C 180,E1 -14871.733,E2 -14871.733} C_VEL
LIN {X 0,Y 339.118,Z 529.779,A -85,B 0,C 180,E1 -14872.707,E2 -14872.707} C_VEL
LIN {X 0,Y 340.849,Z 516.126,A -85,B 0,C 180,E1 -14873.427,E2 -14873.427} C_VEL
LIN {X 0,Y 342.385,Z 495.483,A -85,B 0,C 180,E1 -14874.199,E2 -14874.199} C_VEL
LIN {X 0,Y 345.574,Z 453.56,A -85,B 0,C 180,E1 -14875.655,E2 -14875.655} C_VEL
LIN {X 0,Y 344.728,Z 439.349,A -85,B 0,C 180,E1 -14876.467,E2 -14876.467} C_VEL
LIN {X 0,Y 342.937,Z 425.88,A -85,B 0,C 180,E1 -14877.442,E2 -14877.442} C_VEL
LIN {X 0,Y 340.562,Z 412.766,A -85,B 0,C 180,E1 -14878.574,E2 -14878.574} C_VEL
LIN {X 0,Y 338.419,Z 403.209,A -85,B 0,C 180,E1 -14879.55,E2 -14879.55} C_VEL
LIN {X 0,Y 335.375,Z 396.702,A -85,B 0,C 180,E1 -14880.623,E2 -14880.623} C_VEL
LIN {X 0,Y 334.03,Z 390.258,A -85,B 0,C 180,E1 -14883.166,E2 -14883.166} C_VEL
LIN {X 0,Y 332.832,Z 385.149,A -85,B 0,C 180,E1 -14885.5,E2 -14885.5} C_VEL
LIN {X 0,Y 331.352,Z 380.173,A -85,B 0,C 180,E1 -14888.3,E2 -14888.3} C_VEL
LIN {X 0,Y 330.548,Z 377.622,A -85,B 0,C 180,E1 -14890.055,E2 -14890.055} C_VEL
LIN {X 0,Y 329.319,Z 373.884,A -85,B 0,C 180,E1 -14893.481,E2 -14893.481} C_VEL
LIN {X 0,Y 328.627,Z 371.75,A -85,B 0,C 180,E1 -14896.815,E2 -14896.815} C_VEL
LIN {X 0,Y 328.451,Z 371.23,A -85,B 0,C 180,E1 -14898.498,E2 -14898.498} C_VEL
LIN {X 0,Y 328.445,Z 371.213,A -85,B 0,C 180,E1 -14901.644,E2 -14901.644} C_VEL
LIN {X 0,Y 328.691,Z 372.216,A -85,B 0,C 180,E1 -14904.343,E2 -14904.343} C_VEL
LIN {X 0,Y 329.434,Z 374.776,A -85,B 0,C 180,E1 -14907.867,E2 -14907.867} C_VEL
LIN {X 0,Y 330.43,Z 376.485,A -85,B 0,C 180,E1 -14908.378,E2 -14908.378} C_VEL
LIN {X 0,Y 333.449,Z 379.908,A -85,B 0,C 180,E1 -14909.465,E2 -14909.465} C_VEL
LIN {X 0,Y 337.077,Z 384.809,A -85,B 0,C 180,E1 -14910.686,E2 -14910.686} C_VEL
LIN {X 0,Y 341.366,Z 390.907,A -85,B 0,C 180,E1 -14911.989,E2 -14911.989} C_VEL
LIN {X 0,Y 346.501,Z 399.774,A -85,B 0,C 180,E1 -14913.452,E2 -14913.452} C_VEL
LIN {X 0,Y 348.579,Z 404.083,A -85,B 0,C 180,E1 -14914.033,E2 -14914.033} C_VEL
LIN {X 0,Y 342.875,Z 473.724,A -85,B 0,C 180,E1 -14916.521,E2 -14916.521} C_VEL
LIN {X 0,Y 341.729,Z 487.574,A -85,B 0,C 180,E1 -14917.238,E2 -14917.238} C_VEL
LIN {X 0,Y 340.328,Z 500.673,A -85,B 0,C 180,E1 -14918.179,E2 -14918.179} C_VEL
LIN {X 0,Y 338.629,Z 513.129,A -85,B 0,C 180,E1 -14919.34,E2 -14919.34} C_VEL
LIN {X 0,Y 336.818,Z 524.258,A -85,B 0,C 180,E1 -14920.655,E2 -14920.655} C_VEL
LIN {X 0,Y 335.081,Z 533.404,A -85,B 0,C 180,E1 -14921.979,E2 -14921.979} C_VEL
LIN {X 0,Y 333.088,Z 543.337,A -85,B 0,C 180,E1 -14923.765,E2 -14923.765} C_VEL
LIN {X 0,Y 331.405,Z 551.238,A -85,B 0,C 180,E1 -14925.571,E2 -14925.571} C_VEL
LIN {X 0,Y 330.164,Z 556.652,A -85,B 0,C 180,E1 -14927.085,E2 -14927.085} C_VEL
LIN {X 0,Y 328.909,Z 561.893,A -85,B 0,C 180,E1 -14928.912,E2 -14928.912} C_VEL
LIN {X 0,Y 327.757,Z 565.973,A -85,B 0,C 180,E1 -14930.745,E2 -14930.745} C_VEL
LIN {X 0,Y 326.951,Z 568.933,A -85,B 0,C 180,E1 -14932.59,E2 -14932.59} C_VEL
LIN {X 0,Y 326.541,Z 570.354,A -85,B 0,C 180,E1 -14933.822,E2 -14933.822} C_VEL
LIN {X 0,Y 326.396,Z 571.299,A -85,B 0,C 180,E1 -14935.059,E2 -14935.059} C_VEL
LIN {X 0,Y 326.112,Z 571.823,A -85,B 0,C 180,E1 -14936.293,E2 -14936.293} C_VEL
LIN {X 0,Y 325.736,Z 571.952,A -85,B 0,C 180,E1 -14937.527,E2 -14937.527} C_VEL
LIN {X 0,Y 325.481,Z 571.653,A -85,B 0,C 180,E1 -14938.763,E2 -14938.763} C_VEL
LIN {X 0,Y 325.37,Z 570.875,A -85,B 0,C 180,E1 -14940,E2 -14940} C_VEL
LIN {X 0,Y 325.368,Z 569.675,A -85,B 0,C 180,E1 -14941.238,E2 -14941.238} C_VEL
LIN {X 0,Y 325.402,Z 567.044,A -85,B 0,C 180,E1 -14943.095,E2 -14943.095} C_VEL
LIN {X 0,Y 325.565,Z 563.35,A -85,B 0,C 180,E1 -14944.953,E2 -14944.953} C_VEL
LIN {X 0,Y 325.799,Z 557.616,A -85,B 0,C 180,E1 -14947.11,E2 -14947.11} C_VEL
LIN {X 0,Y 326.155,Z 551.138,A -85,B 0,C 180,E1 -14948.988,E2 -14948.988} C_VEL
LIN {X 0,Y 326.729,Z 543.157,A -85,B 0,C 180,E1 -14950.848,E2 -14950.848} C_VEL
LIN {X 0,Y 327.312,Z 535.031,A -85,B 0,C 180,E1 -14952.399,E2 -14952.399} C_VEL
LIN {X 0,Y 328.199,Z 524.023,A -85,B 0,C 180,E1 -14954.098,E2 -14954.098} C_VEL
LIN {X 0,Y 328.973,Z 512.86,A -85,B 0,C 180,E1 -14955.488,E2 -14955.488} C_VEL
LIN {X 0,Y 329.609,Z 500.991,A -85,B 0,C 180,E1 -14956.665,E2 -14956.665} C_VEL
LIN {X 0,Y 330.285,Z 488.315,A -85,B 0,C 180,E1 -14957.651,E2 -14957.651} C_VEL
LIN {X 0,Y 330.981,Z 474.079,A -85,B 0,C 180,E1 -14958.452,E2 -14958.452} C_VEL
LIN {X 0,Y 331.304,Z 461.004,A -85,B 0,C 180,E1 -14958.955,E2 -14958.955} C_VEL
LIN {X 0,Y 333.41,Z 386.721,A -85,B 0,C 180,E1 -14961.183,E2 -14961.183} C_VEL
LIN {X 0,Y 326.674,Z 365.793,A -85,B 0,C 180,E1 -14962.135,E2 -14962.135} C_VEL
LIN {X 0,Y 326.695,Z 365.787,A -85,B 0,C 180,E1 -14965.483,E2 -14965.483} C_VEL
LIN {X 0,Y 326.666,Z 365.792,A -85,B 0,C 180,E1 -14969.658,E2 -14969.658} C_VEL
LIN {X 0,Y 326.612,Z 365.801,A -85,B 0,C 180,E1 -14974.019,E2 -14974.019} C_VEL
LIN {X 0,Y 326.632,Z 365.795,A -85,B 0,C 180,E1 -14977.238,E2 -14977.238} C_VEL
LIN {X 0,Y 326.582,Z 365.801,A -85,B 0,C 180,E1 -14981.13,E2 -14981.13} C_VEL
LIN {X 0,Y 326.532,Z 365.809,A -85,B 0,C 180,E1 -14984.742,E2 -14984.742} C_VEL
LIN {X 0,Y 326.58,Z 365.807,A -85,B 0,C 180,E1 -14988.153,E2 -14988.153} C_VEL
LIN {X 0,Y 326.628,Z 365.796,A -85,B 0,C 180,E1 -14991.391,E2 -14991.391} C_VEL
LIN {X 0,Y 326.623,Z 365.797,A -85,B 0,C 180,E1 -14994.85,E2 -14994.85} C_VEL
LIN {X 0,Y 326.614,Z 365.798,A -85,B 0,C 180,E1 -14997.455,E2 -14997.455} C_VEL
LIN {X 0,Y 326.652,Z 365.797,A -85,B 0,C 180,E1 -15000.339,E2 -15000.339} C_VEL
LIN {X 0,Y 326.694,Z 365.79,A -85,B 0,C 180,E1 -15004.515,E2 -15004.515} C_VEL
LIN {X 0,Y 326.65,Z 365.795,A -85,B 0,C 180,E1 -15008.544,E2 -15008.544} C_VEL
LIN {X 0,Y 326.747,Z 365.781,A -85,B 0,C 180,E1 -15011.176,E2 -15011.176} C_VEL
LIN {X 0,Y 326.766,Z 365.779,A -85,B 0,C 180,E1 -15015.432,E2 -15015.432} C_VEL
LIN {X 0,Y 326.773,Z 365.778,A -85,B 0,C 180,E1 -15018.838,E2 -15018.838} C_VEL
LIN {X 0,Y 326.96,Z 365.755,A -85,B 0,C 180,E1 -15022.589,E2 -15022.589} C_VEL
LIN {X 0,Y 326.779,Z 365.777,A -85,B 0,C 180,E1 -15025.063,E2 -15025.063} C_VEL
LIN {X 0,Y 327.05,Z 365.745,A -85,B 0,C 180,E1 -15027.535,E2 -15027.535} C_VEL
LIN {X 0,Y 327.219,Z 365.728,A -85,B 0,C 180,E1 -15029.999,E2 -15029.999} C_VEL
LIN {X 0,Y 327.05,Z 365.745,A -85,B 0,C 180,E1 -15032.462,E2 -15032.462} C_VEL
LIN {X 0,Y 326.997,Z 365.753,A -85,B 0,C 180,E1 -15036.168,E2 -15036.168} C_VEL
LIN {X 0,Y 326.914,Z 365.76,A -85,B 0,C 180,E1 -15038.654,E2 -15038.654} C_VEL
LIN {X 0,Y 326.734,Z 365.784,A -85,B 0,C 180,E1 -15042.42,E2 -15042.42} C_VEL
LIN {X 0,Y 326.753,Z 365.78,A -85,B 0,C 180,E1 -15044.956,E2 -15044.956} C_VEL
LIN {X 0,Y 326.731,Z 365.783,A -85,B 0,C 180,E1 -15048.837,E2 -15048.837} C_VEL
LIN {X 0,Y 326.618,Z 365.797,A -85,B 0,C 180,E1 -15052.786,E2 -15052.786} C_VEL
LIN {X 0,Y 326.687,Z 365.791,A -85,B 0,C 180,E1 -15055.482,E2 -15055.482} C_VEL
LIN {X 0,Y 326.658,Z 365.796,A -85,B 0,C 180,E1 -15059.657,E2 -15059.657} C_VEL
LIN {X 0,Y 326.618,Z 365.797,A -85,B 0,C 180,E1 -15062.946,E2 -15062.946} C_VEL
LIN {X 0,Y 326.628,Z 365.796,A -85,B 0,C 180,E1 -15067.045,E2 -15067.045} C_VEL
LIN {X 0,Y 326.629,Z 365.797,A -85,B 0,C 180,E1 -15070.201,E2 -15070.201} C_VEL
LIN {X 0,Y 326.652,Z 365.796,A -85,B 0,C 180,E1 -15073.508,E2 -15073.508} C_VEL
LIN {X 0,Y 326.644,Z 365.794,A -85,B 0,C 180,E1 -15077.013,E2 -15077.013} C_VEL
LIN {X 0,Y 326.638,Z 365.794,A -85,B 0,C 180,E1 -15080.764,E2 -15080.764} C_VEL
LIN {X 0,Y 326.604,Z 365.799,A -85,B 0,C 180,E1 -15084.479,E2 -15084.479} C_VEL
LIN {X 0,Y 326.601,Z 365.803,A -85,B 0,C 180,E1 -15087.455,E2 -15087.455} C_VEL
LIN {X 0,Y 326.639,Z 365.794,A -85,B 0,C 180,E1 -15090.116,E2 -15090.116} C_VEL
LIN {X 0,Y 326.019,Z 365.874,A -85,B 0,C 180,E1 -15091.145,E2 -15091.145} C_VEL
LIN {X 0,Y 323.196,Z 366.23,A -85,B 0,C 180,E1 -15092.82,E2 -15092.82} C_VEL
LIN {X 0,Y 320.756,Z 366.533,A -85,B 0,C 180,E1 -15094.176,E2 -15094.176} C_VEL
LIN {X 0,Y 319.678,Z 366.664,A -85,B 0,C 180,E1 -15095.227,E2 -15095.227} C_VEL
LIN {X 0,Y 319.576,Z 366.674,A -85,B 0,C 180,E1 -15095.583,E2 -15095.583} C_VEL
LIN {X 0,Y 319.606,Z 366.674,A -85,B 0,C 180,E1 -15099.401,E2 -15099.401} C_VEL
LIN {X 0,Y 319.649,Z 366.666,A -85,B 0,C 180,E1 -15102.073,E2 -15102.073} C_VEL
LIN {X 0,Y 319.723,Z 366.658,A -85,B 0,C 180,E1 -15106.008,E2 -15106.008} C_VEL
LIN {X 0,Y 319.75,Z 366.655,A -85,B 0,C 180,E1 -15109.873,E2 -15109.873} C_VEL
LIN {X 0,Y 319.923,Z 366.631,A -85,B 0,C 180,E1 -15112.426,E2 -15112.426} C_VEL
LIN {X 0,Y 319.74,Z 366.655,A -85,B 0,C 180,E1 -15114.956,E2 -15114.956} C_VEL
LIN {X 0,Y 320,Z 366.627,A -85,B 0,C 180,E1 -15117.483,E2 -15117.483} C_VEL
LIN {X 0,Y 320.16,Z 366.603,A -85,B 0,C 180,E1 -15120,E2 -15120} C_VEL
LIN {X 0,Y 319.984,Z 366.623,A -85,B 0,C 180,E1 -15122.518,E2 -15122.518} C_VEL
LIN {X 0,Y 319.946,Z 366.628,A -85,B 0,C 180,E1 -15126.306,E2 -15126.306} C_VEL
LIN {X 0,Y 319.834,Z 366.643,A -85,B 0,C 180,E1 -15128.848,E2 -15128.848} C_VEL
LIN {X 0,Y 319.676,Z 366.662,A -85,B 0,C 180,E1 -15132.7,E2 -15132.7} C_VEL
LIN {X 0,Y 319.69,Z 366.664,A -85,B 0,C 180,E1 -15135.296,E2 -15135.296} C_VEL
LIN {X 0,Y 319.666,Z 366.667,A -85,B 0,C 180,E1 -15139.256,E2 -15139.256} C_VEL
LIN {X 0,Y 319.562,Z 366.681,A -85,B 0,C 180,E1 -15143.32,E2 -15143.32} C_VEL
LIN {X 0,Y 319.61,Z 366.67,A -85,B 0,C 180,E1 -15146.09,E2 -15146.09} C_VEL
LIN {X 0,Y 319.572,Z 366.677,A -85,B 0,C 180,E1 -15148.936,E2 -15148.936} C_VEL
LIN {X 0,Y 319.523,Z 366.682,A -85,B 0,C 180,E1 -15151.863,E2 -15151.863} C_VEL
LIN {X 0,Y 319.574,Z 366.678,A -85,B 0,C 180,E1 -15155.545,E2 -15155.545} C_VEL
LIN {X 0,Y 319.596,Z 366.672,A -85,B 0,C 180,E1 -15158.005,E2 -15158.005} C_VEL
LIN {X 0,Y 319.596,Z 366.674,A -85,B 0,C 180,E1 -15161.614,E2 -15161.614} C_VEL
LIN {X 0,Y 319.64,Z 366.671,A -85,B 0,C 180,E1 -15165.287,E2 -15165.287} C_VEL
LIN {X 0,Y 319.578,Z 366.675,A -85,B 0,C 180,E1 -15168.722,E2 -15168.722} C_VEL
LIN {X 0,Y 319.594,Z 366.672,A -85,B 0,C 180,E1 -15172.341,E2 -15172.341} C_VEL
LIN {X 0,Y 319.559,Z 366.681,A -85,B 0,C 180,E1 -15175.125,E2 -15175.125} C_VEL
LIN {X 0,Y 319.611,Z 366.784,A -85,B 0,C 180,E1 -15177.358,E2 -15177.358} C_VEL
LIN {X 0,Y 322.609,Z 381.294,A -85,B 0,C 180,E1 -15181.048,E2 -15181.048} C_VEL
LIN {X 0,Y 323.796,Z 387.342,A -85,B 0,C 180,E1 -15182.536,E2 -15182.536} C_VEL
LIN {X 0,Y 322.869,Z 397.485,A -85,B 0,C 180,E1 -15184.885,E2 -15184.885} C_VEL
LIN {X 0,Y 321.758,Z 408.21,A -85,B 0,C 180,E1 -15187.317,E2 -15187.317} C_VEL
LIN {X 0,Y 324.506,Z 438.965,A -85,B 0,C 180,E1 -15188.435,E2 -15188.435} C_VEL
LIN {X 0,Y 325.805,Z 450.173,A -85,B 0,C 180,E1 -15188.846,E2 -15188.846} C_VEL
LIN {X 0,Y 323.814,Z 518.937,A -85,B 0,C 180,E1 -15191.043,E2 -15191.043} C_VEL
LIN {X 0,Y 323.044,Z 531.913,A -85,B 0,C 180,E1 -15191.695,E2 -15191.695} C_VEL
LIN {X 0,Y 322.167,Z 544.117,A -85,B 0,C 180,E1 -15192.547,E2 -15192.547} C_VEL
LIN {X 0,Y 321.377,Z 556.196,A -85,B 0,C 180,E1 -15193.649,E2 -15193.649} C_VEL
LIN {X 0,Y 320.493,Z 567.613,A -85,B 0,C 180,E1 -15194.962,E2 -15194.962} C_VEL
LIN {X 0,Y 319.815,Z 577.254,A -85,B 0,C 180,E1 -15196.337,E2 -15196.337} C_VEL
LIN {X 0,Y 319.192,Z 586.413,A -85,B 0,C 180,E1 -15197.928,E2 -15197.928} C_VEL
LIN {X 0,Y 318.675,Z 593.952,A -85,B 0,C 180,E1 -15199.519,E2 -15199.519} C_VEL
LIN {X 0,Y 318.408,Z 601.341,A -85,B 0,C 180,E1 -15201.433,E2 -15201.433} C_VEL
LIN {X 0,Y 318.299,Z 607.592,A -85,B 0,C 180,E1 -15203.514,E2 -15203.514} C_VEL
LIN {X 0,Y 318.269,Z 612.251,A -85,B 0,C 180,E1 -15205.569,E2 -15205.569} C_VEL
LIN {X 0,Y 318.346,Z 615.326,A -85,B 0,C 180,E1 -15207.471,E2 -15207.471} C_VEL
LIN {X 0,Y 318.516,Z 616.773,A -85,B 0,C 180,E1 -15208.737,E2 -15208.737} C_VEL
LIN {X 0,Y 318.491,Z 617.694,A -85,B 0,C 180,E1 -15210.001,E2 -15210.001} C_VEL
LIN {X 0,Y 318.271,Z 618.158,A -85,B 0,C 180,E1 -15211.267,E2 -15211.267} C_VEL
LIN {X 0,Y 318.172,Z 618.196,A -85,B 0,C 180,E1 -15212.533,E2 -15212.533} C_VEL
LIN {X 0,Y 318.01,Z 617.742,A -85,B 0,C 180,E1 -15213.803,E2 -15213.803} C_VEL
LIN {X 0,Y 317.991,Z 615.971,A -85,B 0,C 180,E1 -15215.979,E2 -15215.979} C_VEL
LIN {X 0,Y 318.149,Z 612.739,A -85,B 0,C 180,E1 -15218.257,E2 -15218.257} C_VEL
LIN {X 0,Y 318.539,Z 608.887,A -85,B 0,C 180,E1 -15220.168,E2 -15220.168} C_VEL
LIN {X 0,Y 319.3,Z 603.923,A -85,B 0,C 180,E1 -15222.071,E2 -15222.071} C_VEL
LIN {X 0,Y 320.382,Z 597.732,A -85,B 0,C 180,E1 -15223.965,E2 -15223.965} C_VEL
LIN {X 0,Y 321.838,Z 589.867,A -85,B 0,C 180,E1 -15225.905,E2 -15225.905} C_VEL
LIN {X 0,Y 323.734,Z 580.809,A -85,B 0,C 180,E1 -15227.695,E2 -15227.695} C_VEL
LIN {X 0,Y 325.906,Z 570.428,A -85,B 0,C 180,E1 -15229.364,E2 -15229.364} C_VEL
LIN {X 0,Y 328.171,Z 558.839,A -85,B 0,C 180,E1 -15230.858,E2 -15230.858} C_VEL
LIN {X 0,Y 330.506,Z 545.962,A -85,B 0,C 180,E1 -15232.177,E2 -15232.177} C_VEL
LIN {X 0,Y 332.885,Z 532.252,A -85,B 0,C 180,E1 -15233.238,E2 -15233.238} C_VEL
LIN {X 0,Y 334.87,Z 518.352,A -85,B 0,C 180,E1 -15234.036,E2 -15234.036} C_VEL
LIN {X 0,Y 336.269,Z 503.479,A -85,B 0,C 180,E1 -15234.668,E2 -15234.668} C_VEL
LIN {X 0,Y 340.192,Z 454.401,A -85,B 0,C 180,E1 -15236.43,E2 -15236.43} C_VEL
LIN {X 0,Y 339.521,Z 441.124,A -85,B 0,C 180,E1 -15237.222,E2 -15237.222} C_VEL
LIN {X 0,Y 337.92,Z 427.906,A -85,B 0,C 180,E1 -15238.22,E2 -15238.22} C_VEL
LIN {X 0,Y 335.788,Z 415.431,A -85,B 0,C 180,E1 -15239.355,E2 -15239.355} C_VEL
LIN {X 0,Y 334.232,Z 407.733,A -85,B 0,C 180,E1 -15240.16,E2 -15240.16} C_VEL
LIN {X 0,Y 331.114,Z 401.208,A -85,B 0,C 180,E1 -15241.312,E2 -15241.312} C_VEL
LIN {X 0,Y 328.019,Z 394.934,A -85,B 0,C 180,E1 -15242.616,E2 -15242.616} C_VEL
LIN {X 0,Y 326.619,Z 388.596,A -85,B 0,C 180,E1 -15245.52,E2 -15245.52} C_VEL
LIN {X 0,Y 324.994,Z 382.966,A -85,B 0,C 180,E1 -15248.84,E2 -15248.84} C_VEL
LIN {X 0,Y 323.625,Z 378.697,A -85,B 0,C 180,E1 -15252.317,E2 -15252.317} C_VEL
LIN {X 0,Y 322.695,Z 376.024,A -85,B 0,C 180,E1 -15255.818,E2 -15255.818} C_VEL
LIN {X 0,Y 322.446,Z 375.158,A -85,B 0,C 180,E1 -15257.823,E2 -15257.823} C_VEL
LIN {X 0,Y 322.331,Z 374.838,A -85,B 0,C 180,E1 -15260.779,E2 -15260.779} C_VEL
LIN {X 0,Y 322.488,Z 375.063,A -85,B 0,C 180,E1 -15262.395,E2 -15262.395} C_VEL
LIN {X 0,Y 322.835,Z 376.821,A -85,B 0,C 180,E1 -15265.869,E2 -15265.869} C_VEL
LIN {X 0,Y 325.562,Z 380.322,A -85,B 0,C 180,E1 -15267.185,E2 -15267.185} C_VEL
LIN {X 0,Y 326.959,Z 381.758,A -85,B 0,C 180,E1 -15267.763,E2 -15267.763} C_VEL
LIN {X 0,Y 330.59,Z 386.323,A -85,B 0,C 180,E1 -15269.179,E2 -15269.179} C_VEL
LIN {X 0,Y 333.752,Z 390.687,A -85,B 0,C 180,E1 -15270.302,E2 -15270.302} C_VEL
LIN {X 0,Y 337.722,Z 396.548,A -85,B 0,C 180,E1 -15271.576,E2 -15271.576} C_VEL
LIN {X 0,Y 342.558,Z 405.197,A -85,B 0,C 180,E1 -15273.038,E2 -15273.038} C_VEL
LIN {X 0,Y 343.392,Z 407.034,A -85,B 0,C 180,E1 -15273.293,E2 -15273.293} C_VEL
LIN {X 0,Y 337.375,Z 474.742,A -85,B 0,C 180,E1 -15275.787,E2 -15275.787} C_VEL
LIN {X 0,Y 336.151,Z 488.333,A -85,B 0,C 180,E1 -15276.513,E2 -15276.513} C_VEL
LIN {X 0,Y 334.807,Z 500.074,A -85,B 0,C 180,E1 -15277.361,E2 -15277.361} C_VEL
LIN {X 0,Y 333.114,Z 511.858,A -85,B 0,C 180,E1 -15278.445,E2 -15278.445} C_VEL
LIN {X 0,Y 331.041,Z 523.912,A -85,B 0,C 180,E1 -15279.85,E2 -15279.85} C_VEL
LIN {X 0,Y 329.008,Z 533.936,A -85,B 0,C 180,E1 -15281.312,E2 -15281.312} C_VEL
LIN {X 0,Y 326.861,Z 543.869,A -85,B 0,C 180,E1 -15283.126,E2 -15283.126} C_VEL
LIN {X 0,Y 325.025,Z 551.773,A -85,B 0,C 180,E1 -15284.961,E2 -15284.961} C_VEL
LIN {X 0,Y 323.42,Z 558.165,A -85,B 0,C 180,E1 -15286.811,E2 -15286.811} C_VEL
LIN {X 0,Y 322.086,Z 563.219,A -85,B 0,C 180,E1 -15288.674,E2 -15288.674} C_VEL
LIN {X 0,Y 320.846,Z 567.136,A -85,B 0,C 180,E1 -15290.544,E2 -15290.544} C_VEL
LIN {X 0,Y 319.983,Z 569.934,A -85,B 0,C 180,E1 -15292.427,E2 -15292.427} C_VEL
LIN {X 0,Y 319.542,Z 571.248,A -85,B 0,C 180,E1 -15293.686,E2 -15293.686} C_VEL
LIN {X 0,Y 319.363,Z 572.081,A -85,B 0,C 180,E1 -15294.95,E2 -15294.95} C_VEL
LIN {X 0,Y 319.071,Z 572.528,A -85,B 0,C 180,E1 -15296.211,E2 -15296.211} C_VEL
LIN {X 0,Y 318.675,Z 572.579,A -85,B 0,C 180,E1 -15297.472,E2 -15297.472} C_VEL
LIN {X 0,Y 318.417,Z 572.15,A -85,B 0,C 180,E1 -15298.735,E2 -15298.735} C_VEL
LIN {X 0,Y 318.306,Z 571.292,A -85,B 0,C 180,E1 -15300,E2 -15300} C_VEL
LIN {X 0,Y 318.289,Z 570.019,A -85,B 0,C 180,E1 -15301.265,E2 -15301.265} C_VEL
LIN {X 0,Y 318.312,Z 567.243,A -85,B 0,C 180,E1 -15303.164,E2 -15303.164} C_VEL
LIN {X 0,Y 318.502,Z 563.395,A -85,B 0,C 180,E1 -15305.064,E2 -15305.064} C_VEL
LIN {X 0,Y 318.68,Z 558.083,A -85,B 0,C 180,E1 -15307.057,E2 -15307.057} C_VEL
LIN {X 0,Y 319.028,Z 551.974,A -85,B 0,C 180,E1 -15308.871,E2 -15308.871} C_VEL
LIN {X 0,Y 319.594,Z 544.037,A -85,B 0,C 180,E1 -15310.773,E2 -15310.773} C_VEL
LIN {X 0,Y 320.187,Z 535.955,A -85,B 0,C 180,E1 -15312.357,E2 -15312.357} C_VEL
LIN {X 0,Y 320.927,Z 526.137,A -85,B 0,C 180,E1 -15313.939,E2 -15313.939} C_VEL
LIN {X 0,Y 321.871,Z 514.279,A -85,B 0,C 180,E1 -15315.48,E2 -15315.48} C_VEL
LIN {X 0,Y 322.471,Z 503.362,A -85,B 0,C 180,E1 -15316.621,E2 -15316.621} C_VEL
LIN {X 0,Y 323.211,Z 489.868,A -85,B 0,C 180,E1 -15317.723,E2 -15317.723} C_VEL
LIN {X 0,Y 323.82,Z 476.156,A -85,B 0,C 180,E1 -15318.547,E2 -15318.547} C_VEL
LIN {X 0,Y 324.272,Z 461.67,A -85,B 0,C 180,E1 -15319.136,E2 -15319.136} C_VEL
LIN {X 0,Y 326.419,Z 387.946,A -85,B 0,C 180,E1 -15321.417,E2 -15321.417} C_VEL
LIN {X 0,Y 319.629,Z 366.673,A -85,B 0,C 180,E1 -15322.417,E2 -15322.417} C_VEL
LIN {X 0,Y 319.64,Z 366.669,A -85,B 0,C 180,E1 -15326.087,E2 -15326.087} C_VEL
LIN {X 0,Y 319.594,Z 366.673,A -85,B 0,C 180,E1 -15328.933,E2 -15328.933} C_VEL
LIN {X 0,Y 319.537,Z 366.681,A -85,B 0,C 180,E1 -15331.861,E2 -15331.861} C_VEL
LIN {X 0,Y 319.584,Z 366.673,A -85,B 0,C 180,E1 -15335.542,E2 -15335.542} C_VEL
LIN {X 0,Y 319.578,Z 366.677,A -85,B 0,C 180,E1 -15338.007,E2 -15338.007} C_VEL
LIN {X 0,Y 319.53,Z 366.68,A -85,B 0,C 180,E1 -15341.596,E2 -15341.596} C_VEL
LIN {X 0,Y 319.492,Z 366.684,A -85,B 0,C 180,E1 -15345.256,E2 -15345.256} C_VEL
LIN {X 0,Y 319.533,Z 366.681,A -85,B 0,C 180,E1 -15348.711,E2 -15348.711} C_VEL
LIN {X 0,Y 319.581,Z 366.678,A -85,B 0,C 180,E1 -15352.343,E2 -15352.343} C_VEL
LIN {X 0,Y 319.564,Z 366.676,A -85,B 0,C 180,E1 -15355.122,E2 -15355.122} C_VEL
LIN {X 0,Y 319.57,Z 366.675,A -85,B 0,C 180,E1 -15359.058,E2 -15359.058} C_VEL
LIN {X 0,Y 319.61,Z 366.672,A -85,B 0,C 180,E1 -15362.497,E2 -15362.497} C_VEL
LIN {X 0,Y 319.608,Z 366.67,A -85,B 0,C 180,E1 -15365.303,E2 -15365.303} C_VEL
LIN {X 0,Y 319.6,Z 366.676,A -85,B 0,C 180,E1 -15368.047,E2 -15368.047} C_VEL
LIN {X 0,Y 319.692,Z 366.66,A -85,B 0,C 180,E1 -15370.961,E2 -15370.961} C_VEL
LIN {X 0,Y 319.734,Z 366.655,A -85,B 0,C 180,E1 -15375.275,E2 -15375.275} C_VEL
LIN {X 0,Y 319.755,Z 366.656,A -85,B 0,C 180,E1 -15379.871,E2 -15379.871} C_VEL
LIN {X 0,Y 319.914,Z 366.634,A -85,B 0,C 180,E1 -15382.424,E2 -15382.424} C_VEL
LIN {X 0,Y 319.748,Z 366.652,A -85,B 0,C 180,E1 -15384.955,E2 -15384.955} C_VEL
LIN {X 0,Y 319.994,Z 366.623,A -85,B 0,C 180,E1 -15387.481,E2 -15387.481} C_VEL
LIN {X 0,Y 320.17,Z 366.606,A -85,B 0,C 180,E1 -15389.999,E2 -15389.999} C_VEL
LIN {X 0,Y 319.993,Z 366.623,A -85,B 0,C 180,E1 -15392.516,E2 -15392.516} C_VEL
LIN {X 0,Y 319.953,Z 366.63,A -85,B 0,C 180,E1 -15396.304,E2 -15396.304} C_VEL
LIN {X 0,Y 319.842,Z 366.641,A -85,B 0,C 180,E1 -15398.846,E2 -15398.846} C_VEL
LIN {X 0,Y 319.681,Z 366.661,A -85,B 0,C 180,E1 -15402.698,E2 -15402.698} C_VEL
LIN {X 0,Y 319.698,Z 366.66,A -85,B 0,C 180,E1 -15405.294,E2 -15405.294} C_VEL
LIN {X 0,Y 319.673,Z 366.663,A -85,B 0,C 180,E1 -15409.253,E2 -15409.253} C_VEL
LIN {X 0,Y 319.568,Z 366.676,A -85,B 0,C 180,E1 -15413.318,E2 -15413.318} C_VEL
LIN {X 0,Y 319.632,Z 366.671,A -85,B 0,C 180,E1 -15416.086,E2 -15416.086} C_VEL
LIN {X 0,Y 319.586,Z 366.673,A -85,B 0,C 180,E1 -15418.932,E2 -15418.932} C_VEL
LIN {X 0,Y 319.534,Z 366.685,A -85,B 0,C 180,E1 -15421.859,E2 -15421.859} C_VEL
LIN {X 0,Y 319.576,Z 366.677,A -85,B 0,C 180,E1 -15425.542,E2 -15425.542} C_VEL
LIN {X 0,Y 319.595,Z 366.675,A -85,B 0,C 180,E1 -15428.003,E2 -15428.003} C_VEL
LIN {X 0,Y 319.595,Z 366.676,A -85,B 0,C 180,E1 -15431.611,E2 -15431.611} C_VEL
LIN {X 0,Y 319.639,Z 366.668,A -85,B 0,C 180,E1 -15435.284,E2 -15435.284} C_VEL
LIN {X 0,Y 319.576,Z 366.674,A -85,B 0,C 180,E1 -15438.719,E2 -15438.719} C_VEL
LIN {X 0,Y 319.591,Z 366.673,A -85,B 0,C 180,E1 -15442.338,E2 -15442.338} C_VEL
LIN {X 0,Y 319.552,Z 366.678,A -85,B 0,C 180,E1 -15445.122,E2 -15445.122} C_VEL
LIN {X 0,Y 319.562,Z 366.677,A -85,B 0,C 180,E1 -15449.057,E2 -15449.057} C_VEL
LIN {X 0,Y 319.608,Z 366.67,A -85,B 0,C 180,E1 -15452.498,E2 -15452.498} C_VEL
LIN {X 0,Y 319.576,Z 366.674,A -85,B 0,C 180,E1 -15455.583,E2 -15455.583} C_VEL
LIN {X 0,Y 318.878,Z 366.762,A -85,B 0,C 180,E1 -15456.634,E2 -15456.634} C_VEL
LIN {X 0,Y 316.055,Z 367.113,A -85,B 0,C 180,E1 -15458.348,E2 -15458.348} C_VEL
LIN {X 0,Y 313.694,Z 367.411,A -85,B 0,C 180,E1 -15459.736,E2 -15459.736} C_VEL
LIN {X 0,Y 312.693,Z 367.532,A -85,B 0,C 180,E1 -15460.81,E2 -15460.81} C_VEL
LIN {X 0,Y 312.616,Z 367.542,A -85,B 0,C 180,E1 -15461.173,E2 -15461.173} C_VEL
LIN {X 0,Y 312.685,Z 367.537,A -85,B 0,C 180,E1 -15465.686,E2 -15465.686} C_VEL
LIN {X 0,Y 312.694,Z 367.536,A -85,B 0,C 180,E1 -15469.642,E2 -15469.642} C_VEL
LIN {X 0,Y 312.862,Z 367.511,A -85,B 0,C 180,E1 -15472.254,E2 -15472.254} C_VEL
LIN {X 0,Y 312.71,Z 367.53,A -85,B 0,C 180,E1 -15474.842,E2 -15474.842} C_VEL
LIN {X 0,Y 312.943,Z 367.505,A -85,B 0,C 180,E1 -15477.426,E2 -15477.426} C_VEL
LIN {X 0,Y 313.112,Z 367.481,A -85,B 0,C 180,E1 -15480,E2 -15480} C_VEL
LIN {X 0,Y 312.93,Z 367.502,A -85,B 0,C 180,E1 -15482.575,E2 -15482.575} C_VEL
LIN {X 0,Y 312.904,Z 367.505,A -85,B 0,C 180,E1 -15486.448,E2 -15486.448} C_VEL
LIN {X 0,Y 312.779,Z 367.523,A -85,B 0,C 180,E1 -15489.05,E2 -15489.05} C_VEL
LIN {X 0,Y 312.628,Z 367.541,A -85,B 0,C 180,E1 -15492.992,E2 -15492.992} C_VEL
LIN {X 0,Y 312.629,Z 367.543,A -85,B 0,C 180,E1 -15495.65,E2 -15495.65} C_VEL
LIN {X 0,Y 312.621,Z 367.544,A -85,B 0,C 180,E1 -15499.237,E2 -15499.237} C_VEL
LIN {X 0,Y 312.537,Z 367.552,A -85,B 0,C 180,E1 -15502.79,E2 -15502.79} C_VEL
LIN {X 0,Y 312.588,Z 367.545,A -85,B 0,C 180,E1 -15505.934,E2 -15505.934} C_VEL
LIN {X 0,Y 312.53,Z 367.554,A -85,B 0,C 180,E1 -15509.652,E2 -15509.652} C_VEL
LIN {X 0,Y 312.512,Z 367.556,A -85,B 0,C 180,E1 -15513.69,E2 -15513.69} C_VEL
LIN {X 0,Y 312.548,Z 367.554,A -85,B 0,C 180,E1 -15517.382,E2 -15517.382} C_VEL
LIN {X 0,Y 312.529,Z 367.553,A -85,B 0,C 180,E1 -15520.703,E2 -15520.703} C_VEL
LIN {X 0,Y 312.589,Z 367.544,A -85,B 0,C 180,E1 -15524.185,E2 -15524.185} C_VEL
LIN {X 0,Y 312.551,Z 367.55,A -85,B 0,C 180,E1 -15527.905,E2 -15527.905} C_VEL
LIN {X 0,Y 312.554,Z 367.549,A -85,B 0,C 180,E1 -15531.906,E2 -15531.906} C_VEL
LIN {X 0,Y 312.505,Z 367.556,A -85,B 0,C 180,E1 -15535.792,E2 -15535.792} C_VEL
LIN {X 0,Y 312.583,Z 367.587,A -85,B 0,C 180,E1 -15537.129,E2 -15537.129} C_VEL
LIN {X 0,Y 315.666,Z 382.637,A -85,B 0,C 180,E1 -15541.039,E2 -15541.039} C_VEL
LIN {X 0,Y 316.786,Z 388.648,A -85,B 0,C 180,E1 -15542.551,E2 -15542.551} C_VEL
LIN {X 0,Y 315.358,Z 401.901,A -85,B 0,C 180,E1 -15545.679,E2 -15545.679} C_VEL
LIN {X 0,Y 314.799,Z 407.552,A -85,B 0,C 180,E1 -15547.004,E2 -15547.004} C_VEL
LIN {X 0,Y 316.804,Z 432.143,A -85,B 0,C 180,E1 -15547.928,E2 -15547.928} C_VEL
LIN {X 0,Y 318.761,Z 451.48,A -85,B 0,C 180,E1 -15548.653,E2 -15548.653} C_VEL
LIN {X 0,Y 316.814,Z 518.282,A -85,B 0,C 180,E1 -15550.861,E2 -15550.861} C_VEL
LIN {X 0,Y 316.022,Z 531.201,A -85,B 0,C 180,E1 -15551.526,E2 -15551.526} C_VEL
LIN {X 0,Y 315.223,Z 542.465,A -85,B 0,C 180,E1 -15552.317,E2 -15552.317} C_VEL
LIN {X 0,Y 314.415,Z 554.734,A -85,B 0,C 180,E1 -15553.443,E2 -15553.443} C_VEL
LIN {X 0,Y 313.56,Z 565.882,A -85,B 0,C 180,E1 -15554.73,E2 -15554.73} C_VEL
LIN {X 0,Y 312.779,Z 576.085,A -85,B 0,C 180,E1 -15556.19,E2 -15556.19} C_VEL
LIN {X 0,Y 312.091,Z 586.186,A -85,B 0,C 180,E1 -15557.979,E2 -15557.979} C_VEL
LIN {X 0,Y 311.606,Z 593.683,A -85,B 0,C 180,E1 -15559.607,E2 -15559.607} C_VEL
LIN {X 0,Y 311.359,Z 601.002,A -85,B 0,C 180,E1 -15561.565,E2 -15561.565} C_VEL
LIN {X 0,Y 311.262,Z 606.753,A -85,B 0,C 180,E1 -15563.519,E2 -15563.519} C_VEL
LIN {X 0,Y 311.223,Z 611.165,A -85,B 0,C 180,E1 -15565.468,E2 -15565.468} C_VEL
LIN {X 0,Y 311.292,Z 614.376,A -85,B 0,C 180,E1 -15567.414,E2 -15567.414} C_VEL
LIN {X 0,Y 311.47,Z 615.921,A -85,B 0,C 180,E1 -15568.709,E2 -15568.709} C_VEL
LIN {X 0,Y 311.445,Z 616.945,A -85,B 0,C 180,E1 -15570.001,E2 -15570.001} C_VEL
LIN {X 0,Y 311.209,Z 617.467,A -85,B 0,C 180,E1 -15571.296,E2 -15571.296} C_VEL
LIN {X 0,Y 311.097,Z 617.569,A -85,B 0,C 180,E1 -15572.591,E2 -15572.591} C_VEL
LIN {X 0,Y 310.932,Z 617.23,A -85,B 0,C 180,E1 -15573.89,E2 -15573.89} C_VEL
LIN {X 0,Y 310.896,Z 615.791,A -85,B 0,C 180,E1 -15575.928,E2 -15575.928} C_VEL
LIN {X 0,Y 311.086,Z 612.506,A -85,B 0,C 180,E1 -15578.446,E2 -15578.446} C_VEL
LIN {X 0,Y 311.525,Z 608.811,A -85,B 0,C 180,E1 -15580.399,E2 -15580.399} C_VEL
LIN {X 0,Y 312.354,Z 604.008,A -85,B 0,C 180,E1 -15582.344,E2 -15582.344} C_VEL
LIN {X 0,Y 313.712,Z 596.901,A -85,B 0,C 180,E1 -15584.599,E2 -15584.599} C_VEL
LIN {X 0,Y 315.336,Z 589.217,A -85,B 0,C 180,E1 -15586.53,E2 -15586.53} C_VEL
LIN {X 0,Y 317.453,Z 579.975,A -85,B 0,C 180,E1 -15588.391,E2 -15588.391} C_VEL
LIN {X 0,Y 319.746,Z 569.62,A -85,B 0,C 180,E1 -15590.088,E2 -15590.088} C_VEL
LIN {X 0,Y 322.203,Z 558.081,A -85,B 0,C 180,E1 -15591.599,E2 -15591.599} C_VEL
LIN {X 0,Y 324.664,Z 545.327,A -85,B 0,C 180,E1 -15592.934,E2 -15592.934} C_VEL
LIN {X 0,Y 327.397,Z 530.719,A -85,B 0,C 180,E1 -15594.072,E2 -15594.072} C_VEL
LIN {X 0,Y 329.583,Z 516.059,A -85,B 0,C 180,E1 -15594.908,E2 -15594.908} C_VEL
LIN {X 0,Y 331.019,Z 500.92,A -85,B 0,C 180,E1 -15595.549,E2 -15595.549} C_VEL
LIN {X 0,Y 334.973,Z 455.64,A -85,B 0,C 180,E1 -15597.227,E2 -15597.227} C_VEL
LIN {X 0,Y 334.518,Z 443.518,A -85,B 0,C 180,E1 -15597.971,E2 -15597.971} C_VEL
LIN {X 0,Y 332.976,Z 429.595,A -85,B 0,C 180,E1 -15599.075,E2 -15599.075} C_VEL
LIN {X 0,Y 330.986,Z 416.976,A -85,B 0,C 180,E1 -15600.286,E2 -15600.286} C_VEL
LIN {X 0,Y 329.97,Z 412.043,A -85,B 0,C 180,E1 -15600.846,E2 -15600.846} C_VEL
LIN {X 0,Y 327.393,Z 406.302,A -85,B 0,C 180,E1 -15601.894,E2 -15601.894} C_VEL
LIN {X 0,Y 324.247,Z 400.016,A -85,B 0,C 180,E1 -15603.254,E2 -15603.254} C_VEL
LIN {X 0,Y 320.717,Z 393.184,A -85,B 0,C 180,E1 -15605.015,E2 -15605.015} C_VEL
LIN {X 0,Y 319.255,Z 387.778,A -85,B 0,C 180,E1 -15608.054,E2 -15608.054} C_VEL
LIN {X 0,Y 318.53,Z 385.3,A -85,B 0,C 180,E1 -15609.782,E2 -15609.782} C_VEL
LIN {X 0,Y 317.226,Z 381.477,A -85,B 0,C 180,E1 -15613.378,E2 -15613.378} C_VEL
LIN {X 0,Y 316.55,Z 379.431,A -85,B 0,C 180,E1 -15616.507,E2 -15616.507} C_VEL
LIN {X 0,Y 316.31,Z 378.66,A -85,B 0,C 180,E1 -15619.065,E2 -15619.065} C_VEL
LIN {X 0,Y 316.326,Z 378.623,A -85,B 0,C 180,E1 -15621.531,E2 -15621.531} C_VEL
LIN {X 0,Y 316.453,Z 379.09,A -85,B 0,C 180,E1 -15623.204,E2 -15623.204} C_VEL
LIN {X 0,Y 319.142,Z 382.399,A -85,B 0,C 180,E1 -15624.951,E2 -15624.951} C_VEL
LIN {X 0,Y 320.635,Z 383.754,A -85,B 0,C 180,E1 -15625.722,E2 -15625.722} C_VEL
LIN {X 0,Y 323.466,Z 387.135,A -85,B 0,C 180,E1 -15627.099,E2 -15627.099} C_VEL
LIN {X 0,Y 327.502,Z 392.327,A -85,B 0,C 180,E1 -15628.791,E2 -15628.791} C_VEL
LIN {X 0,Y 330.444,Z 396.525,A -85,B 0,C 180,E1 -15629.89,E2 -15629.89} C_VEL
LIN {X 0,Y 334.096,Z 402.137,A -85,B 0,C 180,E1 -15631.145,E2 -15631.145} C_VEL
LIN {X 0,Y 338.308,Z 409.895,A -85,B 0,C 180,E1 -15632.499,E2 -15632.499} C_VEL
LIN {X 0,Y 331.969,Z 476.317,A -85,B 0,C 180,E1 -15635.033,E2 -15635.033} C_VEL
LIN {X 0,Y 330.513,Z 490.607,A -85,B 0,C 180,E1 -15635.837,E2 -15635.837} C_VEL
